C09107=1052.158,191.230,408.588,171.579,35.261,156.618
C09108=1052.153,190.981,408.612,171.577,35.259,156.618
C09109=1052.147,190.732,408.636,171.575,35.257,156.617
C09110=1052.140,190.448,408.663,171.573,35.253,156.616
C09111=1052.134,190.163,408.691,171.570,35.251,156.616
C09112=1052.127,189.880,408.719,171.567,35.248,156.615
C09113=1052.121,189.595,408.746,171.564,35.245,156.615
C09114=1052.114,189.346,408.770,171.562,35.242,156.614
C09115=1052.109,189.098,408.794,171.560,35.240,156.614
C09116=1052.102,188.849,408.818,171.558,35.237,156.613
C09117=1052.097,188.600,408.843,171.555,35.235,156.613
C09118=1052.091,188.352,408.866,171.553,35.232,156.612
C09119=1052.085,188.102,408.890,171.551,35.229,156.612
C09120=1052.079,187.854,408.914,171.549,35.227,156.611
C09121=1052.073,187.605,408.938,171.547,35.224,156.611
C09122=1052.067,187.356,408.962,171.543,35.222,156.611
C09123=1052.062,187.108,408.986,171.541,35.219,156.610
C09124=1052.055,186.859,409.010,171.539,35.217,156.610
C09125=1052.049,186.610,409.033,171.537,35.214,156.609
C09126=1052.044,186.361,409.058,171.535,35.212,156.609
C09127=1052.037,186.112,409.082,171.533,35.209,156.608
C09128=1052.032,185.864,409.106,171.530,35.206,156.608
C09129=1052.026,185.615,409.130,171.528,35.204,156.607
C09130=1052.021,185.365,409.153,171.526,35.201,156.607
C09131=1052.014,185.117,409.177,171.524,35.199,156.606
C09132=1052.009,184.869,409.201,171.522,35.196,156.606
C09133=1052.003,184.620,409.225,171.518,35.194,156.605
C09134=1051.997,184.371,409.248,171.516,35.191,156.605
C09135=1051.992,184.122,409.273,171.514,35.189,156.604
C09136=1051.985,183.873,409.297,171.512,35.187,156.604
C09137=1051.979,183.624,409.320,171.510,35.184,156.603
C09138=1051.973,183.375,409.344,171.508,35.182,156.603
C09139=1051.967,183.126,409.367,171.505,35.179,156.602
C09140=1051.961,182.878,409.390,171.503,35.177,156.602
C09141=1051.954,182.628,409.413,171.501,35.175,156.602
C09142=1051.948,182.380,409.437,171.499,35.172,156.601
C09143=1051.942,182.131,409.460,171.496,35.170,156.601
C09144=1051.935,181.883,409.484,171.494,35.167,156.600
C09145=1051.930,181.634,409.506,171.491,35.165,156.600
C09146=1051.923,181.385,409.530,171.489,35.163,156.599
C09147=1051.917,181.136,409.553,171.487,35.160,156.599
C09148=1051.911,180.888,409.577,171.485,35.158,156.599
C09149=1051.905,180.638,409.600,171.483,35.155,156.598
C09150=1051.899,180.390,409.624,171.481,35.154,156.598
C09151=1051.893,180.141,409.647,171.478,35.151,156.597
C09152=1051.886,179.892,409.671,171.476,35.149,156.597
C09153=1051.881,179.643,409.694,171.474,35.146,156.596
C09154=1051.875,179.395,409.718,171.472,35.144,156.596
C09155=1051.868,179.145,409.741,171.469,35.142,156.595
C09156=1051.862,178.896,409.763,171.467,35.139,156.595
C09157=1051.856,178.648,409.787,171.464,35.137,156.595
C09158=1051.849,178.399,409.810,171.462,35.134,156.594
C09159=1051.844,178.150,409.833,171.460,35.132,156.594
C09160=1051.838,177.901,409.857,171.458,35.130,156.593
C09161=1051.832,177.653,409.880,171.456,35.127,156.593
C09162=1051.825,177.404,409.904,171.454,35.125,156.592
C09163=1051.820,177.155,409.927,171.451,35.122,156.592
C09164=1051.814,176.906,409.950,171.449,35.120,156.592
C09165=1051.808,176.656,409.973,171.447,35.118,156.591
C09166=1051.801,176.408,409.996,171.445,35.115,156.591
C09167=1051.795,176.159,410.019,171.443,35.113,156.590
C09168=1051.789,175.910,410.042,171.441,35.111,156.590
C09169=1051.783,175.662,410.066,171.438,35.109,156.589
C09170=1051.777,175.413,410.089,171.436,35.106,156.589
C09171=1051.771,175.164,410.112,171.434,35.104,156.588
C09172=1051.765,174.915,410.135,171.432,35.102,156.588
C09173=1051.759,174.666,410.159,171.430,35.099,156.588
C09174=1051.752,174.381,410.185,171.427,35.096,156.587
C09175=1051.746,174.097,410.211,171.424,35.094,156.587
C09176=1051.739,173.813,410.237,171.422,35.091,156.586
C09177=1051.732,173.527,410.264,171.419,35.089,156.586
C09178=1051.725,173.279,410.286,171.417,35.086,156.585
C09179=1051.719,173.030,410.310,171.415,35.084,156.585
C09180=1051.714,172.781,410.333,171.413,35.081,156.584
C09181=1051.707,172.532,410.356,171.410,35.079,156.584
C09182=1051.702,172.283,410.379,171.408,35.077,156.583
C09183=1051.696,172.034,410.402,171.406,35.074,156.583
C09184=1051.689,171.786,410.424,171.404,35.072,156.583
C09185=1051.684,171.537,410.447,171.402,35.069,156.582
C09186=1051.678,171.288,410.470,171.400,35.067,156.582
C09187=1051.672,171.039,410.494,171.399,35.065,156.581
C09188=1051.666,170.791,410.517,171.396,35.062,156.581
C09189=1051.660,170.541,410.540,171.394,35.060,156.580
C09190=1051.653,170.292,410.563,171.392,35.058,156.580
C09191=1051.648,170.043,410.586,171.390,35.056,156.580
C09192=1051.642,169.795,410.608,171.388,35.053,156.579
C09193=1051.636,169.546,410.631,171.386,35.051,156.579
C09194=1051.630,169.297,410.654,171.383,35.049,156.578
C09195=1051.625,169.048,410.677,171.381,35.046,156.578
C09196=1051.618,168.799,410.700,171.379,35.044,156.577
C09197=1051.612,168.550,410.723,171.377,35.041,156.577
C09198=1051.607,168.302,410.746,171.375,35.039,156.577
C09199=1051.601,168.053,410.769,171.373,35.037,156.576
C09200=1051.595,167.804,410.791,171.370,35.034,156.576
C09201=1051.589,167.555,410.814,171.368,35.032,156.575
C09202=1051.583,167.306,410.837,171.366,35.030,156.575
C09203=1051.577,167.057,410.860,171.364,35.027,156.574
C09204=1051.572,166.808,410.883,171.362,35.025,156.574
C09205=1051.566,166.560,410.906,171.360,35.022,156.573
C09206=1051.559,166.311,410.928,171.358,35.020,156.573
C09207=1051.554,166.061,410.950,171.355,35.018,156.573
C09208=1051.548,165.813,410.973,171.353,35.015,156.572
C09209=1051.543,165.564,410.996,171.351,35.013,156.572
C09210=1051.537,165.315,411.019,171.350,35.011,156.571
C09211=1051.530,165.066,411.041,171.348,35.009,156.571
C09212=1051.525,164.817,411.064,171.346,35.006,156.570
C09213=1051.519,164.568,411.087,171.343,35.004,156.570
C09214=1051.513,164.319,411.109,171.341,35.002,156.570
C09215=1051.507,164.070,411.132,171.339,34.999,156.569
C09216=1051.501,163.821,411.155,171.337,34.997,156.569
C09217=1051.496,163.572,411.178,171.335,34.994,156.568
C09218=1051.490,163.324,411.201,171.333,34.992,156.568
C09219=1051.483,163.075,411.223,171.331,34.990,156.567
C09220=1051.478,162.825,411.245,171.328,34.987,156.567
C09221=1051.472,162.577,411.268,171.327,34.985,156.566
C09222=1051.466,162.328,411.291,171.325,34.983,156.566
C09223=1051.460,162.079,411.313,171.323,34.980,156.566
C09224=1051.455,161.830,411.336,171.321,34.978,156.565
C09225=1051.449,161.581,411.359,171.319,34.975,156.565
C09226=1051.444,161.332,411.381,171.317,34.974,156.564
C09227=1051.438,161.083,411.403,171.314,34.971,156.564
C09228=1051.432,160.834,411.426,171.312,34.969,156.564
C09229=1051.426,160.585,411.449,171.310,34.967,156.563
C09230=1051.420,160.336,411.470,171.308,34.964,156.563
C09231=1051.414,160.087,411.493,171.307,34.962,156.562
C09232=1051.408,159.839,411.516,171.305,34.960,156.562
C09233=1051.402,159.590,411.537,171.303,34.957,156.561
C09234=1051.396,159.341,411.560,171.300,34.955,156.561
C09235=1051.390,159.091,411.582,171.298,34.953,156.561
C09236=1051.384,158.843,411.605,171.296,34.951,156.560
C09237=1051.377,158.594,411.627,171.294,34.948,156.560
C09238=1051.371,158.309,411.652,171.292,34.946,156.559
C09239=1051.364,158.023,411.678,171.290,34.943,156.559
C09240=1051.357,157.739,411.703,171.288,34.941,156.558
C09241=1051.350,157.454,411.728,171.284,34.938,156.558
C09242=1051.344,157.205,411.751,171.283,34.937,156.558
C09243=1051.338,156.956,411.773,171.281,34.934,156.557
C09244=1051.332,156.707,411.795,171.279,34.932,156.557
C09245=1051.326,156.457,411.817,171.277,34.930,156.556
C09246=1051.320,156.209,411.840,171.275,34.927,156.556
C09247=1051.314,155.960,411.861,171.273,34.925,156.556
C09248=1051.308,155.711,411.884,171.270,34.923,156.555
C09249=1051.302,155.462,411.906,171.268,34.921,156.555
C09250=1051.296,155.213,411.927,171.266,34.918,156.554
C09251=1051.291,154.964,411.950,171.265,34.916,156.554
C09252=1051.284,154.715,411.972,171.263,34.914,156.554
C09253=1051.278,154.466,411.994,171.261,34.912,156.553
C09254=1051.273,154.217,412.016,171.259,34.909,156.553
C09255=1051.266,153.968,412.038,171.257,34.908,156.552
C09256=1051.260,153.719,412.060,171.254,34.905,156.552
C09257=1051.254,153.471,412.082,171.252,34.903,156.552
C09258=1051.248,153.221,412.103,171.251,34.901,156.551
C09259=1051.242,152.972,412.126,171.249,34.899,156.551
C09260=1051.236,152.723,412.148,171.247,34.896,156.550
C09261=1051.230,152.474,412.169,171.245,34.894,156.550
C09262=1051.224,152.225,412.192,171.243,34.892,156.550
C09263=1051.218,151.977,412.213,171.240,34.890,156.549
C09264=1051.213,151.727,412.235,171.238,34.887,156.549
C09265=1051.206,151.479,412.258,171.237,34.886,156.548
C09266=1051.200,151.230,412.279,171.235,34.883,156.548
C09267=1051.194,150.980,412.301,171.233,34.881,156.548
C09268=1051.188,150.731,412.323,171.231,34.879,156.547
C09269=1051.183,150.483,412.345,171.229,34.877,156.547
C09270=1051.176,150.234,412.367,171.227,34.874,156.546
C09271=1051.170,149.985,412.388,171.224,34.872,156.546
C09272=1051.164,149.735,412.410,171.223,34.870,156.546
C09273=1051.158,149.487,412.432,171.221,34.868,156.545
C09274=1051.152,149.238,412.454,171.219,34.866,156.545
C09275=1051.147,148.989,412.476,171.217,34.863,156.544
C09276=1051.140,148.740,412.498,171.215,34.862,156.544
C09277=1051.134,148.490,412.519,171.213,34.859,156.544
C09278=1051.129,148.242,412.540,171.212,34.857,156.543
C09279=1051.122,147.993,412.563,171.209,34.855,156.543
C09280=1051.116,147.744,412.584,171.207,34.853,156.542
C09281=1051.110,147.495,412.606,171.205,34.850,156.542
C09282=1051.104,147.246,412.627,171.203,34.848,156.542
C09283=1051.098,146.997,412.649,171.201,34.846,156.541
C09284=1051.092,146.748,412.671,171.200,34.844,156.541
C09285=1051.086,146.499,412.692,171.198,34.842,156.541
C09286=1051.080,146.250,412.714,171.196,34.840,156.540
C09287=1051.074,146.001,412.735,171.193,34.838,156.540
C09288=1051.068,145.752,412.757,171.191,34.836,156.539
C09289=1051.062,145.503,412.778,171.189,34.833,156.539
C09290=1051.056,145.253,412.800,171.188,34.831,156.539
C09291=1051.050,145.005,412.821,171.186,34.829,156.538
C09292=1051.044,144.756,412.843,171.184,34.827,156.538
C09293=1051.038,144.506,412.865,171.182,34.825,156.537
C09294=1051.032,144.258,412.886,171.180,34.823,156.537
C09295=1051.026,144.009,412.907,171.178,34.821,156.537
C09296=1051.020,143.760,412.929,171.176,34.819,156.536
C09297=1051.014,143.510,412.951,171.174,34.816,156.536
C09298=1051.007,143.262,412.971,171.172,34.814,156.536
C09299=1051.001,143.013,412.993,171.170,34.812,156.535
C09300=1050.995,142.764,413.015,171.169,34.810,156.535
C09301=1050.990,142.515,413.036,171.167,34.808,156.534
C09302=1050.982,142.229,413.061,171.165,34.805,156.534
C09303=1050.976,141.944,413.086,171.162,34.803,156.534
C09304=1050.969,141.659,413.110,171.160,34.800,156.533
C09305=1050.963,141.373,413.134,171.158,34.798,156.533
C09306=1050.956,141.124,413.156,171.156,34.796,156.532
C09307=1050.950,140.875,413.177,171.154,34.794,156.532
C09308=1050.945,140.626,413.199,171.152,34.791,156.531
C09309=1050.938,140.377,413.220,171.150,34.790,156.531
C09310=1050.932,140.129,413.241,171.149,34.787,156.531
C09311=1050.926,139.879,413.262,171.146,34.785,156.530
C09312=1050.920,139.630,413.284,171.144,34.783,156.530
C09313=1050.915,139.381,413.305,171.142,34.781,156.530
C09314=1050.908,139.132,413.326,171.140,34.779,156.529
C09315=1050.902,138.883,413.348,171.139,34.777,156.529
C09316=1050.896,138.634,413.368,171.137,34.774,156.528
C09317=1050.890,138.385,413.390,171.135,34.772,156.528
C09318=1050.884,138.136,413.411,171.133,34.771,156.528
C09319=1050.878,137.888,413.432,171.131,34.768,156.527
C09320=1050.872,137.638,413.453,171.129,34.766,156.527
C09321=1050.866,137.389,413.475,171.127,34.764,156.527
C09322=1050.860,137.140,413.496,171.125,34.762,156.526
C09323=1050.853,136.891,413.517,171.123,34.760,156.526
C09324=1050.848,136.642,413.537,171.122,34.758,156.525
C09325=1050.842,136.393,413.559,171.120,34.756,156.525
C09326=1050.835,136.144,413.580,171.118,34.753,156.525
C09327=1050.830,135.895,413.601,171.116,34.752,156.524
C09328=1050.823,135.646,413.622,171.114,34.750,156.524
C09329=1050.817,135.397,413.643,171.112,34.747,156.524
C09330=1050.811,135.148,413.664,171.110,34.745,156.523
C09331=1050.805,134.898,413.686,171.108,34.743,156.523
C09332=1050.799,134.650,413.705,171.107,34.741,156.522
C09333=1050.793,134.400,413.727,171.105,34.739,156.522
C09334=1050.787,134.152,413.748,171.103,34.737,156.522
C09335=1050.782,133.902,413.769,171.101,34.734,156.521
C09336=1050.775,133.654,413.790,171.100,34.733,156.521
C09337=1050.769,133.404,413.811,171.097,34.731,156.521
C09338=1050.763,133.156,413.832,171.095,34.729,156.520
C09339=1050.757,132.907,413.853,171.093,34.726,156.520
C09340=1050.751,132.657,413.874,171.092,34.724,156.519
C09341=1050.745,132.409,413.895,171.090,34.722,156.519
C09342=1050.739,132.159,413.916,171.088,34.720,156.519
C09343=1050.733,131.910,413.937,171.086,34.718,156.518
C09344=1050.727,131.661,413.957,171.085,34.716,156.518
C09345=1050.721,131.412,413.979,171.083,34.713,156.518
C09346=1050.715,131.163,413.999,171.080,34.712,156.517
C09347=1050.709,130.914,414.020,171.078,34.710,156.517
C09348=1050.702,130.665,414.041,171.077,34.708,156.517
C09349=1050.697,130.415,414.061,171.075,34.706,156.516
C09350=1050.690,130.167,414.082,171.073,34.704,156.516
C09351=1050.684,129.917,414.102,171.071,34.701,156.515
C09352=1050.678,129.669,414.124,171.069,34.699,156.515
C09353=1050.672,129.419,414.144,171.068,34.698,156.515
C09354=1050.665,129.171,414.165,171.066,34.696,156.514
C09355=1050.659,128.921,414.186,171.064,34.694,156.514
C09356=1050.653,128.672,414.206,171.061,34.691,156.514
C09357=1050.647,128.423,414.227,171.060,34.689,156.513
C09358=1050.641,128.174,414.248,171.058,34.687,156.513
C09359=1050.635,127.925,414.267,171.056,34.685,156.513
C09360=1050.628,127.676,414.289,171.054,34.684,156.512
C09361=1050.622,127.427,414.309,171.053,34.682,156.512
C09362=1050.616,127.177,414.329,171.051,34.679,156.512
C09363=1050.610,126.929,414.351,171.049,34.677,156.511
C09364=1050.604,126.679,414.371,171.048,34.675,156.511
C09365=1050.598,126.430,414.391,171.046,34.673,156.511
C09366=1050.591,126.145,414.415,171.043,34.671,156.510
C09367=1050.584,125.860,414.438,171.041,34.669,156.510
C09368=1050.577,125.574,414.462,171.039,34.666,156.509
C09369=1050.570,125.289,414.486,171.037,34.664,156.509
C09370=1050.564,125.039,414.507,171.035,34.662,156.508
C09371=1050.558,124.790,414.526,171.033,34.660,156.508
C09372=1050.551,124.541,414.547,171.032,34.658,156.508
C09373=1050.546,124.292,414.568,171.030,34.656,156.507
C09374=1050.539,124.043,414.588,171.028,34.654,156.507
C09375=1050.533,123.794,414.608,171.026,34.652,156.507
C09376=1050.528,123.545,414.629,171.024,34.650,156.506
C09377=1050.521,123.295,414.649,171.022,34.648,156.506
C09378=1050.515,123.047,414.670,171.020,34.645,156.506
C09379=1050.509,122.797,414.691,171.019,34.643,156.505
C09380=1050.503,122.548,414.711,171.017,34.642,156.505
C09381=1050.497,122.299,414.731,171.015,34.640,156.505
C09382=1050.491,122.050,414.752,171.014,34.638,156.504
C09383=1050.485,121.801,414.772,171.012,34.635,156.504
C09384=1050.478,121.552,414.793,171.009,34.633,156.503
C09385=1050.473,121.303,414.813,171.007,34.631,156.503
C09386=1050.467,121.054,414.833,171.006,34.629,156.503
C09387=1050.461,120.805,414.853,171.004,34.627,156.502
C09388=1050.455,120.556,414.873,171.002,34.625,156.502
C09389=1050.449,120.306,414.894,171.001,34.623,156.502
C09390=1050.443,120.057,414.914,170.999,34.621,156.501
C09391=1050.437,119.808,414.934,170.997,34.619,156.501
C09392=1050.431,119.559,414.955,170.996,34.617,156.501
C09393=1050.425,119.310,414.975,170.994,34.615,156.500
C09394=1050.419,119.061,414.995,170.991,34.613,156.500
C09395=1050.413,118.812,415.017,170.990,34.611,156.500
C09396=1050.407,118.563,415.037,170.988,34.608,156.499
C09397=1050.401,118.314,415.057,170.986,34.606,156.499
C09398=1050.394,118.065,415.077,170.985,34.605,156.498
C09399=1050.389,117.815,415.098,170.983,34.603,156.498
C09400=1050.383,117.567,415.118,170.981,34.600,156.498
C09401=1050.376,117.317,415.138,170.979,34.598,156.497
C09402=1050.371,117.068,415.158,170.978,34.596,156.497
C09403=1050.365,116.819,415.178,170.976,34.594,156.497
C09404=1050.359,116.570,415.198,170.973,34.592,156.496
C09405=1050.352,116.321,415.219,170.972,34.590,156.496
C09406=1050.347,116.072,415.239,170.970,34.588,156.495
C09407=1050.341,115.823,415.259,170.968,34.586,156.495
C09408=1050.335,115.573,415.279,170.967,34.584,156.495
C09409=1050.329,115.324,415.299,170.965,34.582,156.494
C09410=1050.324,115.075,415.319,170.963,34.580,156.494
C09411=1050.318,114.826,415.339,170.962,34.578,156.494
C09412=1050.311,114.577,415.360,170.960,34.575,156.493
C09413=1050.305,114.328,415.380,170.958,34.573,156.493
C09414=1050.300,114.079,415.400,170.957,34.571,156.493
C09415=1050.294,113.830,415.420,170.954,34.569,156.492
C09416=1050.287,113.580,415.440,170.952,34.567,156.492
C09417=1050.281,113.331,415.460,170.951,34.565,156.491
C09418=1050.276,113.082,415.480,170.949,34.563,156.491
C09419=1050.270,112.833,415.500,170.947,34.561,156.491
C09420=1050.263,112.584,415.520,170.946,34.559,156.490
C09421=1050.257,112.335,415.540,170.944,34.557,156.490
C09422=1050.251,112.086,415.560,170.942,34.555,156.490
C09423=1050.245,111.836,415.579,170.941,34.554,156.489
C09424=1050.239,111.587,415.599,170.939,34.551,156.489
C09425=1050.233,111.338,415.619,170.936,34.549,156.489
C09426=1050.227,111.089,415.639,170.935,34.547,156.488
C09427=1050.220,110.839,415.659,170.933,34.545,156.488
C09428=1050.214,110.591,415.679,170.931,34.543,156.488
C09429=1050.208,110.342,415.699,170.930,34.541,156.487
C09430=1050.201,110.056,415.721,170.928,34.539,156.487
C09431=1050.194,109.770,415.744,170.926,34.537,156.487
C09432=1050.187,109.484,415.766,170.924,34.534,156.486
C09433=1050.180,109.198,415.789,170.922,34.532,156.486
C09434=1050.173,108.950,415.809,170.920,34.530,156.485
C09435=1050.167,108.701,415.829,170.919,34.529,156.485
C09436=1050.162,108.452,415.848,170.916,34.526,156.485
C09437=1050.155,108.202,415.868,170.914,34.524,156.484
C09438=1050.149,107.953,415.888,170.913,34.522,156.484
C09439=1050.143,107.704,415.907,170.911,34.520,156.484
C09440=1050.137,107.455,415.927,170.909,34.518,156.483
C09441=1050.131,107.206,415.947,170.908,34.516,156.483
C09442=1050.124,106.956,415.966,170.906,34.514,156.483
C09443=1050.118,106.708,415.986,170.904,34.513,156.482
C09444=1050.113,106.458,416.006,170.903,34.511,156.482
C09445=1050.107,106.209,416.026,170.901,34.509,156.482
C09446=1050.101,105.960,416.045,170.899,34.506,156.481
C09447=1050.094,105.711,416.064,170.897,34.504,156.481
C09448=1050.088,105.462,416.084,170.895,34.502,156.481
C09449=1050.082,105.212,416.104,170.893,34.500,156.480
C09450=1050.076,104.964,416.124,170.892,34.498,156.480
C09451=1050.070,104.714,416.143,170.890,34.497,156.480
C09452=1050.064,104.465,416.163,170.888,34.495,156.479
C09453=1050.057,104.216,416.182,170.887,34.493,156.479
C09454=1050.051,103.967,416.202,170.885,34.491,156.479
C09455=1050.046,103.717,416.221,170.884,34.488,156.478
C09456=1050.040,103.468,416.241,170.882,34.486,156.478
C09457=1050.034,103.219,416.260,170.880,34.484,156.477
C09458=1050.028,102.970,416.280,170.878,34.482,156.477
C09459=1050.022,102.721,416.299,170.876,34.481,156.477
C09460=1050.016,102.472,416.319,170.874,34.479,156.476
C09461=1050.009,102.222,416.338,170.873,34.477,156.476
C09462=1050.003,101.973,416.358,170.871,34.475,156.476
C09463=1049.998,101.724,416.378,170.869,34.472,156.475
C09464=1049.991,101.475,416.397,170.868,34.470,156.475
C09465=1049.985,101.226,416.416,170.866,34.468,156.475
C09466=1049.979,100.977,416.436,170.864,34.466,156.474
C09467=1049.973,100.728,416.455,170.863,34.464,156.474
C09468=1049.967,100.479,416.474,170.861,34.463,156.474
C09469=1049.961,100.230,416.494,170.860,34.461,156.473
C09470=1049.955,99.980,416.514,170.857,34.459,156.473
C09471=1049.948,99.731,416.532,170.855,34.457,156.473
C09472=1049.942,99.482,416.552,170.854,34.455,156.472
C09473=1049.936,99.233,416.571,170.852,34.453,156.472
C09474=1049.930,98.983,416.590,170.850,34.451,156.472
C09475=1049.923,98.735,416.610,170.849,34.449,156.471
C09476=1049.918,98.485,416.629,170.847,34.447,156.471
C09477=1049.911,98.236,416.647,170.845,34.445,156.471
C09478=1049.905,97.986,416.667,170.844,34.443,156.470
C09479=1049.899,97.737,416.687,170.842,34.441,156.470
C09480=1049.893,97.488,416.706,170.840,34.439,156.470
C09481=1049.887,97.239,416.725,170.839,34.437,156.469
C09482=1049.881,96.989,416.744,170.836,34.436,156.469
C09483=1049.875,96.741,416.764,170.834,34.434,156.469
C09484=1049.868,96.492,416.782,170.833,34.432,156.468
C09485=1049.862,96.242,416.801,170.831,34.429,156.468
C09486=1049.856,95.993,416.820,170.830,34.427,156.468
C09487=1049.850,95.744,416.840,170.828,34.425,156.467
C09488=1049.844,95.495,416.859,170.826,34.423,156.467
C09489=1049.838,95.246,416.878,170.825,34.421,156.467
C09490=1049.832,94.996,416.897,170.823,34.419,156.466
C09491=1049.826,94.747,416.916,170.821,34.418,156.466
C09492=1049.820,94.498,416.936,170.820,34.416,156.466
C09493=1049.813,94.249,416.954,170.818,34.414,156.465
C09494=1049.808,94.014,416.972,170.817,34.412,156.465
C09495=1049.802,93.780,416.990,170.814,34.410,156.465
C09496=1049.797,93.545,417.008,170.813,34.408,156.464
C09497=1049.790,93.311,417.026,170.811,34.407,156.464
C09498=1049.784,93.076,417.044,170.809,34.405,156.464
C09499=1049.779,92.842,417.063,170.808,34.403,156.463
C09500=1049.773,92.608,417.080,170.806,34.401,156.463
C09501=1049.768,92.374,417.098,170.805,34.399,156.463
C09502=1049.761,92.124,417.117,170.803,34.397,156.462
C09503=1049.756,91.875,417.136,170.802,34.395,156.462
C09504=1049.749,91.626,417.155,170.800,34.393,156.462
C09505=1049.744,91.376,417.174,170.798,34.391,156.461
C09506=1049.737,91.127,417.193,170.797,34.389,156.461
C09507=1049.731,90.878,417.212,170.795,34.387,156.461
C09508=1049.725,90.629,417.231,170.793,34.385,156.460
C09509=1049.719,90.379,417.250,170.791,34.383,156.460
C09510=1049.711,90.064,417.274,170.789,34.381,156.460
C09511=1049.703,89.749,417.298,170.787,34.378,156.459
C09512=1049.695,89.433,417.321,170.785,34.376,156.459
C09513=1049.687,89.119,417.345,170.783,34.374,156.458
C09514=1049.681,88.870,417.364,170.781,34.372,156.458
C09515=1049.675,88.620,417.383,170.779,34.370,156.458
C09516=1049.669,88.371,417.401,170.778,34.368,156.457
C09517=1049.663,88.122,417.420,170.776,34.366,156.457
C09518=1049.656,87.873,417.439,170.774,34.364,156.457
C09519=1049.650,87.624,417.458,170.773,34.362,156.456
C09520=1049.644,87.374,417.476,170.770,34.360,156.456
C09521=1049.638,87.125,417.495,170.769,34.358,156.456
C09522=1049.631,86.876,417.513,170.767,34.356,156.456
C09523=1049.626,86.626,417.532,170.765,34.354,156.455
C09524=1049.619,86.377,417.551,170.764,34.352,156.455
C09525=1049.613,86.128,417.570,170.762,34.350,156.455
C09526=1049.606,85.879,417.588,170.760,34.349,156.454
C09527=1049.601,85.629,417.608,170.759,34.347,156.454
C09528=1049.594,85.380,417.626,170.757,34.345,156.454
C09529=1049.588,85.131,417.644,170.756,34.343,156.453
C09530=1049.582,84.881,417.663,170.754,34.341,156.453
C09531=1049.577,84.633,417.682,170.752,34.339,156.453
C09532=1049.570,84.384,417.700,170.751,34.337,156.452
C09533=1049.564,84.134,417.719,170.749,34.335,156.452
C09534=1049.557,83.885,417.738,170.746,34.333,156.452
C09535=1049.551,83.636,417.756,170.745,34.331,156.451
C09536=1049.546,83.386,417.775,170.743,34.329,156.451
C09537=1049.539,83.137,417.793,170.742,34.327,156.451
C09538=1049.533,82.888,417.812,170.740,34.325,156.450
C09539=1049.527,82.638,417.830,170.738,34.323,156.450
C09540=1049.521,82.390,417.848,170.737,34.321,156.450
C09541=1049.515,82.140,417.868,170.735,34.319,156.449
C09542=1049.509,81.891,417.886,170.733,34.318,156.449
C09543=1049.502,81.642,417.905,170.732,34.316,156.449
C09544=1049.496,81.392,417.923,170.730,34.314,156.448
C09545=1049.490,81.143,417.941,170.729,34.312,156.448
C09546=1049.484,80.894,417.961,170.727,34.310,156.448
C09547=1049.479,80.645,417.978,170.724,34.308,156.447
C09548=1049.472,80.396,417.997,170.723,34.306,156.447
C09549=1049.466,80.146,418.016,170.721,34.304,156.447
C09550=1049.459,79.897,418.034,170.720,34.302,156.446
C09551=1049.454,79.647,418.053,170.718,34.300,156.446
C09552=1049.448,79.399,418.071,170.716,34.298,156.446
C09553=1049.442,79.150,418.090,170.715,34.296,156.445
C09554=1049.436,78.900,418.108,170.713,34.294,156.445
C09555=1049.429,78.651,418.126,170.712,34.292,156.445
C09556=1049.423,78.401,418.144,170.710,34.290,156.444
C09557=1049.417,78.152,418.163,170.708,34.288,156.444
C09558=1049.410,77.866,418.184,170.706,34.286,156.444
C09559=1049.403,77.581,418.205,170.705,34.285,156.443
C09560=1049.396,77.296,418.226,170.703,34.282,156.443
C09561=1049.388,77.009,418.247,170.700,34.280,156.443
C09562=1049.382,76.760,418.265,170.698,34.278,156.442
C09563=1049.376,76.511,418.283,170.697,34.276,156.442
C09564=1049.370,76.262,418.301,170.695,34.274,156.442
C09565=1049.364,76.012,418.320,170.693,34.272,156.441
C09566=1049.358,75.763,418.338,170.692,34.270,156.441
C09567=1049.351,75.514,418.356,170.690,34.268,156.441
C09568=1049.346,75.265,418.374,170.688,34.267,156.440
C09569=1049.339,75.015,418.393,170.687,34.265,156.440
C09570=1049.333,74.766,418.411,170.685,34.263,156.440
C09571=1049.327,74.517,418.429,170.684,34.261,156.439
C09572=1049.321,74.267,418.447,170.682,34.259,156.439
C09573=1049.315,74.018,418.465,170.680,34.257,156.439
C09574=1049.309,73.769,418.483,170.679,34.255,156.438
C09575=1049.302,73.520,418.502,170.677,34.253,156.438
C09576=1049.295,73.270,418.519,170.675,34.251,156.438
C09577=1049.290,73.022,418.538,170.673,34.250,156.437
C09578=1049.284,72.772,418.556,170.671,34.248,156.437
C09579=1049.277,72.523,418.574,170.670,34.246,156.437
C09580=1049.271,72.273,418.592,170.668,34.244,156.436
C09581=1049.265,72.024,418.610,170.666,34.242,156.436
C09582=1049.259,71.775,418.628,170.665,34.240,156.436
C09583=1049.253,71.525,418.646,170.663,34.238,156.436
C09584=1049.247,71.277,418.665,170.662,34.237,156.435
C09585=1049.241,71.027,418.683,170.660,34.235,156.435
C09586=1049.234,70.778,418.700,170.658,34.233,156.435
C09587=1049.228,70.528,418.719,170.657,34.231,156.434
C09588=1049.222,70.279,418.736,170.655,34.229,156.434
C09589=1049.216,70.030,418.754,170.653,34.227,156.434
C09590=1049.210,69.781,418.773,170.652,34.225,156.433
C09591=1049.204,69.532,418.790,170.650,34.223,156.433
C09592=1049.198,69.282,418.808,170.648,34.221,156.433
C09593=1049.191,69.033,418.826,170.646,34.220,156.432
C09594=1049.185,68.783,418.844,170.644,34.218,156.432
C09595=1049.179,68.534,418.862,170.643,34.216,156.432
C09596=1049.173,68.285,418.880,170.641,34.214,156.431
C09597=1049.166,68.036,418.898,170.640,34.212,156.431
C09598=1049.160,67.787,418.915,170.638,34.210,156.431
C09599=1049.154,67.537,418.933,170.636,34.208,156.431
C09600=1049.148,67.288,418.952,170.635,34.206,156.430
C09601=1049.142,67.039,418.969,170.633,34.204,156.430
C09602=1049.135,66.789,418.987,170.631,34.203,156.430
C09603=1049.129,66.540,419.005,170.630,34.201,156.429
C09604=1049.123,66.291,419.022,170.628,34.199,156.429
C09605=1049.117,66.042,419.040,170.627,34.197,156.429
C09606=1049.111,65.792,419.058,170.625,34.195,156.428
C09607=1049.105,65.543,419.076,170.623,34.193,156.428
C09608=1049.098,65.293,419.093,170.621,34.191,156.428
C09609=1049.092,65.044,419.112,170.619,34.190,156.427
C09610=1049.086,64.795,419.129,170.617,34.188,156.427
C09611=1049.079,64.546,419.147,170.616,34.186,156.427
C09612=1049.073,64.296,419.165,170.614,34.184,156.427
C09613=1049.068,64.047,419.182,170.613,34.182,156.426
C09614=1049.061,63.798,419.200,170.611,34.180,156.426
C09615=1049.055,63.548,419.217,170.609,34.179,156.426
C09616=1049.048,63.298,419.235,170.608,34.177,156.425
C09617=1049.042,63.049,419.252,170.606,34.175,156.425
C09618=1049.035,62.800,419.270,170.604,34.173,156.425
C09619=1049.028,62.551,419.288,170.603,34.171,156.424
C09620=1049.023,62.302,419.305,170.601,34.169,156.424
C09621=1049.016,62.053,419.323,170.599,34.167,156.424
C09622=1049.009,61.767,419.343,170.597,34.165,156.424
C09623=1049.002,61.481,419.363,170.596,34.164,156.423
C09624=1048.994,61.194,419.383,170.594,34.162,156.423
C09625=1048.987,60.908,419.403,170.592,34.160,156.423
C09626=1048.981,60.660,419.420,170.589,34.158,156.422
C09627=1048.975,60.410,419.438,170.588,34.156,156.422
C09628=1048.968,60.160,419.455,170.586,34.154,156.422
C09629=1048.962,59.912,419.472,170.584,34.152,156.421
C09630=1048.956,59.662,419.490,170.583,34.150,156.421
C09631=1048.949,59.413,419.507,170.581,34.148,156.421
C09632=1048.943,59.163,419.525,170.579,34.146,156.420
C09633=1048.937,58.914,419.542,170.578,34.145,156.420
C09634=1048.930,58.665,419.559,170.576,34.143,156.420
C09635=1048.924,58.416,419.577,170.574,34.141,156.420
C09636=1048.917,58.166,419.595,170.573,34.139,156.419
C09637=1048.912,57.917,419.612,170.571,34.137,156.419
C09638=1048.905,57.668,419.629,170.569,34.136,156.419
C09639=1048.899,57.419,419.647,170.568,34.134,156.418
C09640=1048.893,57.169,419.664,170.566,34.132,156.418
C09641=1048.886,56.920,419.681,170.565,34.130,156.418
C09642=1048.881,56.670,419.699,170.563,34.128,156.417
C09643=1048.874,56.421,419.716,170.561,34.127,156.417
C09644=1048.868,56.172,419.733,170.560,34.125,156.417
C09645=1048.861,55.922,419.751,170.557,34.123,156.417
C09646=1048.855,55.673,419.768,170.555,34.121,156.416
C09647=1048.849,55.424,419.786,170.554,34.120,156.416
C09648=1048.843,55.175,419.803,170.552,34.118,156.416
C09649=1048.836,54.925,419.819,170.550,34.116,156.415
C09650=1048.831,54.676,419.837,170.549,34.114,156.415
C09651=1048.824,54.426,419.854,170.547,34.112,156.415
C09652=1048.818,54.177,419.872,170.546,34.110,156.414
C09653=1048.811,53.928,419.889,170.544,34.109,156.414
C09654=1048.805,53.679,419.905,170.542,34.107,156.414
C09655=1048.799,53.429,419.923,170.541,34.105,156.414
C09656=1048.793,53.180,419.940,170.539,34.103,156.413
C09657=1048.786,52.931,419.958,170.537,34.101,156.413
C09658=1048.781,52.682,419.975,170.536,34.099,156.413
C09659=1048.774,52.432,419.992,170.534,34.097,156.412
C09660=1048.769,52.183,420.009,170.532,34.095,156.412
C09661=1048.762,51.933,420.027,170.531,34.093,156.412
C09662=1048.755,51.684,420.044,170.529,34.092,156.411
C09663=1048.750,51.434,420.061,170.528,34.090,156.411
C09664=1048.743,51.185,420.078,170.525,34.088,156.411
C09665=1048.737,50.936,420.095,170.523,34.086,156.411
C09666=1048.731,50.686,420.112,170.522,34.084,156.410
C09667=1048.725,50.438,420.129,170.520,34.083,156.410
C09668=1048.718,50.188,420.146,170.518,34.081,156.410
C09669=1048.713,49.938,420.163,170.517,34.079,156.409
C09670=1048.706,49.689,420.181,170.515,34.077,156.409
C09671=1048.700,49.440,420.197,170.513,34.075,156.409
C09672=1048.694,49.190,420.215,170.512,34.073,156.408
C09673=1048.688,48.941,420.232,170.510,34.072,156.408
C09674=1048.682,48.692,420.249,170.509,34.070,156.408
C09675=1048.676,48.442,420.266,170.507,34.068,156.408
C09676=1048.670,48.193,420.283,170.505,34.066,156.407
C09677=1048.663,47.944,420.301,170.504,34.064,156.407
C09678=1048.657,47.694,420.317,170.502,34.063,156.407
C09679=1048.651,47.446,420.334,170.500,34.061,156.406
C09680=1048.645,47.196,420.351,170.499,34.059,156.406
C09681=1048.639,46.947,420.368,170.497,34.057,156.406
C09682=1048.633,46.698,420.385,170.495,34.055,156.405
C09683=1048.626,46.448,420.402,170.494,34.053,156.405
C09684=1048.621,46.199,420.419,170.491,34.051,156.405
C09685=1048.614,45.949,420.436,170.490,34.049,156.405
C09686=1048.607,45.663,420.456,170.488,34.047,156.404
C09687=1048.601,45.376,420.475,170.486,34.045,156.404
C09688=1048.593,45.091,420.495,170.484,34.043,156.403
C09689=1048.586,44.804,420.514,170.482,34.041,156.403
C09690=1048.581,44.555,420.531,170.480,34.039,156.403
C09691=1048.575,44.306,420.548,170.479,34.037,156.402
C09692=1048.568,44.056,420.565,170.477,34.035,156.402
C09693=1048.562,43.807,420.581,170.476,34.033,156.402
C09694=1048.556,43.558,420.599,170.474,34.031,156.402
C09695=1048.550,43.308,420.615,170.472,34.030,156.401
C09696=1048.544,43.059,420.632,170.471,34.028,156.401
C09697=1048.537,42.809,420.649,170.469,34.026,156.401
C09698=1048.531,42.560,420.666,170.467,34.024,156.400
C09699=1048.525,42.311,420.682,170.466,34.023,156.400
C09700=1048.518,42.061,420.699,170.464,34.021,156.400
C09701=1048.512,41.812,420.716,170.462,34.019,156.400
C09702=1048.506,41.563,420.732,170.461,34.017,156.399
C09703=1048.499,41.313,420.749,170.459,34.015,156.399
C09704=1048.494,41.064,420.766,170.457,34.013,156.399
C09705=1048.488,40.814,420.782,170.455,34.012,156.398
C09706=1048.481,40.565,420.800,170.453,34.010,156.398
C09707=1048.475,40.316,420.816,170.451,34.008,156.398
C09708=1048.469,40.066,420.832,170.450,34.006,156.397
C09709=1048.462,39.817,420.850,170.448,34.005,156.397
C09710=1048.457,39.567,420.866,170.446,34.003,156.397
C09711=1048.451,39.318,420.882,170.445,34.001,156.397
C09712=1048.444,39.069,420.899,170.443,33.999,156.396
C09713=1048.438,38.819,420.916,170.441,33.997,156.396
C09714=1048.432,38.570,420.932,170.440,33.995,156.396
C09715=1048.426,38.321,420.949,170.438,33.993,156.395
C09716=1048.420,38.072,420.965,170.436,33.992,156.395
C09717=1048.413,37.822,420.982,170.435,33.990,156.395
C09718=1048.407,37.572,420.998,170.433,33.988,156.395
C09719=1048.401,37.324,421.015,170.431,33.986,156.394
C09720=1048.394,37.074,421.032,170.430,33.985,156.394
C09721=1048.388,36.824,421.048,170.428,33.983,156.394
C09722=1048.382,36.575,421.064,170.426,33.982,156.394
C09723=1048.375,36.326,421.081,170.425,33.980,156.393
C09724=1048.369,36.076,421.097,170.423,33.978,156.393
C09725=1048.363,35.827,421.114,170.421,33.976,156.393
C09726=1048.357,35.578,421.130,170.420,33.974,156.392
C09727=1048.350,35.328,421.146,170.418,33.972,156.392
C09728=1048.344,35.078,421.163,170.416,33.971,156.392
C09729=1048.338,34.830,421.180,170.414,33.969,156.392
C09730=1048.332,34.581,421.195,170.412,33.968,156.391
C09731=1048.325,34.331,421.212,170.410,33.966,156.391
C09732=1048.319,34.081,421.228,170.408,33.964,156.391
C09733=1048.313,33.832,421.244,170.407,33.962,156.391
C09734=1048.307,33.583,421.261,170.405,33.960,156.390
C09735=1048.300,33.333,421.277,170.403,33.958,156.390
C09736=1048.294,33.083,421.293,170.402,33.957,156.390
C09737=1048.288,32.835,421.310,170.400,33.955,156.389
C09738=1048.282,32.585,421.326,170.398,33.954,156.389
C09739=1048.275,32.335,421.343,170.397,33.952,156.389
C09740=1048.269,32.086,421.359,170.395,33.950,156.389
C09741=1048.262,31.837,421.375,170.393,33.948,156.388
C09742=1048.257,31.588,421.391,170.392,33.946,156.388
C09743=1048.251,31.338,421.407,170.390,33.944,156.388
C09744=1048.244,31.088,421.424,170.388,33.943,156.387
C09745=1048.238,30.839,421.440,170.387,33.941,156.387
C09746=1048.231,30.590,421.456,170.385,33.939,156.387
C09747=1048.225,30.340,421.472,170.383,33.938,156.387
C09748=1048.219,30.091,421.488,170.382,33.936,156.386
C09749=1048.214,29.842,421.505,170.380,33.934,156.386
C09750=1048.206,29.556,421.523,170.378,33.932,156.386
C09751=1048.199,29.269,421.542,170.376,33.930,156.385
C09752=1048.191,28.983,421.560,170.374,33.928,156.385
C09753=1048.185,28.696,421.580,170.372,33.926,156.385
C09754=1048.178,28.447,421.595,170.370,33.924,156.385
C09755=1048.172,28.197,421.611,170.368,33.922,156.384
C09756=1048.166,27.948,421.627,170.366,33.921,156.384
C09757=1048.159,27.698,421.643,170.364,33.919,156.384
C09758=1048.153,27.449,421.659,170.363,33.917,156.383
C09759=1048.146,27.200,421.675,170.361,33.916,156.383
C09760=1048.140,26.951,421.691,170.359,33.914,156.383
C09761=1048.135,26.701,421.708,170.357,33.912,156.383
C09762=1048.128,26.452,421.723,170.356,33.910,156.382
C09763=1048.122,26.203,421.740,170.354,33.909,156.382
C09764=1048.115,25.953,421.756,170.352,33.907,156.382
C09765=1048.109,25.703,421.771,170.351,33.906,156.382
C09766=1048.103,25.454,421.787,170.349,33.904,156.381
C09767=1048.096,25.205,421.803,170.347,33.902,156.381
C09768=1048.090,24.955,421.819,170.345,33.900,156.381
C09769=1048.084,24.706,421.835,170.344,33.898,156.380
C09770=1048.078,24.457,421.851,170.342,33.897,156.380
C09771=1048.072,24.207,421.867,170.340,33.895,156.380
C09772=1048.065,23.957,421.883,170.339,33.894,156.380
C09773=1048.059,23.708,421.899,170.337,33.892,156.379
C09774=1048.052,23.459,421.915,170.335,33.890,156.379
C09775=1048.047,23.209,421.930,170.333,33.888,156.379
C09776=1048.040,22.960,421.946,170.332,33.887,156.379
C09777=1048.034,22.711,421.962,170.330,33.885,156.378
C09778=1048.028,22.461,421.978,170.328,33.884,156.378
C09779=1048.021,22.212,421.994,170.327,33.882,156.378
C09780=1048.016,21.962,422.010,170.325,33.880,156.378
C09781=1048.009,21.713,422.025,170.323,33.878,156.377
C09782=1048.003,21.464,422.042,170.321,33.876,156.377
C09783=1047.997,21.214,422.056,170.320,33.875,156.377
C09784=1047.990,20.964,422.073,170.318,33.873,156.377
C09785=1047.983,20.715,422.089,170.316,33.872,156.376
C09786=1047.977,20.466,422.105,170.315,33.870,156.376
C09787=1047.971,20.216,422.120,170.312,33.868,156.376
C09788=1047.965,19.967,422.136,170.310,33.866,156.375
C09789=1047.958,19.718,422.152,170.308,33.865,156.375
C09790=1047.953,19.468,422.167,170.307,33.863,156.375
C09791=1047.946,19.219,422.183,170.305,33.862,156.375
C09792=1047.940,18.969,422.199,170.303,33.860,156.374
C09793=1047.934,18.720,422.214,170.301,33.858,156.374
C09794=1047.928,18.470,422.231,170.300,33.856,156.374
C09795=1047.921,18.221,422.245,170.298,33.855,156.374
C09796=1047.915,17.972,422.261,170.296,33.853,156.373
C09797=1047.909,17.722,422.277,170.294,33.852,156.373
C09798=1047.902,17.473,422.292,170.293,33.850,156.373
C09799=1047.896,17.223,422.309,170.291,33.848,156.373
C09800=1047.890,16.974,422.324,170.289,33.846,156.372
C09801=1047.883,16.725,422.339,170.288,33.845,156.372
C09802=1047.878,16.475,422.355,170.286,33.843,156.372
C09803=1047.871,16.226,422.370,170.284,33.841,156.372
C09804=1047.865,15.976,422.386,170.282,33.839,156.371
C09805=1047.859,15.727,422.402,170.281,33.838,156.371
C09806=1047.852,15.477,422.417,170.279,33.836,156.371
C09807=1047.846,15.228,422.433,170.277,33.835,156.371
C09808=1047.840,14.978,422.448,170.275,33.833,156.370
C09809=1047.833,14.729,422.463,170.274,33.831,156.370
C09810=1047.828,14.479,422.479,170.272,33.830,156.370
C09811=1047.821,14.230,422.495,170.270,33.828,156.370
C09812=1047.815,13.980,422.510,170.268,33.827,156.369
C09813=1047.809,13.731,422.526,170.267,33.825,156.369
C09814=1047.801,13.446,422.544,170.265,33.823,156.369
C09815=1047.794,13.161,422.561,170.262,33.821,156.369
C09816=1047.787,12.876,422.579,170.260,33.819,156.368
C09817=1047.779,12.591,422.596,170.258,33.818,156.368
C09818=1047.773,12.341,422.611,170.257,33.816,156.368
C09819=1047.766,12.091,422.626,170.255,33.815,156.368
C09820=1047.760,11.843,422.641,170.253,33.813,156.367
C09821=1047.754,11.593,422.656,170.251,33.811,156.367
C09822=1047.747,11.344,422.671,170.250,33.810,156.367
C09823=1047.741,11.094,422.688,170.248,33.808,156.367
C09824=1047.735,10.845,422.702,170.246,33.806,156.366
C09825=1047.728,10.596,422.718,170.244,33.805,156.366
C09826=1047.722,10.346,422.733,170.241,33.803,156.366
C09827=1047.716,10.096,422.748,170.240,33.802,156.366
C09828=1047.709,9.847,422.763,170.238,33.800,156.365
C09829=1047.703,9.598,422.779,170.236,33.798,156.365
C09830=1047.697,9.348,422.794,170.234,33.797,156.365
C09831=1047.691,9.098,422.809,170.233,33.796,156.365
C09832=1047.684,8.849,422.825,170.231,33.794,156.364
C09833=1047.677,8.599,422.840,170.229,33.792,156.364
C09834=1047.671,8.350,422.855,170.227,33.791,156.364
C09835=1047.665,8.101,422.869,170.225,33.789,156.364
C09836=1047.659,7.852,422.885,170.224,33.787,156.363
C09837=1047.652,7.602,422.900,170.222,33.786,156.363
C09838=1047.647,7.352,422.915,170.220,33.784,156.363
C09839=1047.640,7.103,422.930,170.218,33.783,156.363
C09840=1047.633,6.853,422.946,170.217,33.781,156.363
C09841=1047.627,6.604,422.961,170.215,33.779,156.362
C09842=1047.621,6.354,422.976,170.213,33.778,156.362
C09843=1047.614,6.105,422.991,170.211,33.777,156.362
C09844=1047.609,5.856,423.005,170.209,33.774,156.362
C09845=1047.602,5.607,423.021,170.208,33.773,156.361
C09846=1047.595,5.357,423.036,170.206,33.771,156.361
C09847=1047.589,5.107,423.051,170.204,33.770,156.361
C09848=1047.583,4.857,423.067,170.202,33.768,156.361
C09849=1047.577,4.608,423.081,170.200,33.766,156.360
C09850=1047.571,4.359,423.096,170.199,33.765,156.360
C09851=1047.565,4.110,423.112,170.197,33.764,156.360
C09852=1047.558,3.860,423.127,170.195,33.762,156.360
C09853=1047.552,3.610,423.142,170.193,33.760,156.359
C09854=1047.545,3.361,423.157,170.191,33.759,156.359
C09855=1047.540,3.112,423.171,170.190,33.757,156.359
C09856=1047.533,2.862,423.186,170.188,33.756,156.359
C09857=1047.527,2.612,423.201,170.186,33.754,156.359
C09858=1047.521,2.363,423.216,170.184,33.752,156.358
C09859=1047.514,2.113,423.231,170.182,33.751,156.358
C09860=1047.509,1.864,423.247,170.181,33.749,156.358
C09861=1047.502,1.615,423.262,170.179,33.747,156.358
C09862=1047.496,1.365,423.277,170.177,33.746,156.357
C09863=1047.490,1.115,423.292,170.175,33.745,156.357
C09864=1047.484,0.866,423.306,170.173,33.743,156.357
C09865=1047.477,0.617,423.321,170.172,33.741,156.357
C09866=1047.471,0.367,423.336,170.170,33.740,156.356
C09867=1047.465,0.117,423.351,170.168,33.738,156.356
C09868=1047.459,-0.131,423.366,170.166,33.736,156.356
C09869=1047.453,-0.381,423.381,170.164,33.735,156.356
C09870=1047.446,-0.631,423.396,170.163,33.733,156.355
C09871=1047.440,-0.880,423.410,170.161,33.732,156.355
C09872=1047.434,-1.129,423.425,170.159,33.730,156.355
C09873=1047.428,-1.379,423.440,170.157,33.728,156.355
C09874=1047.421,-1.629,423.455,170.155,33.727,156.354
C09875=1047.415,-1.878,423.470,170.154,33.725,156.354
C09876=1047.409,-2.127,423.484,170.152,33.724,156.354
C09877=1047.403,-2.377,423.499,170.150,33.722,156.354
C09878=1047.396,-2.661,423.516,170.147,33.720,156.353
C09879=1047.390,-2.943,423.533,170.145,33.718,156.353
C09880=1047.382,-3.226,423.549,170.143,33.717,156.353
C09881=1047.375,-3.509,423.566,170.141,33.715,156.353
C09882=1047.369,-3.760,423.581,170.139,33.713,156.352
C09883=1047.363,-4.008,423.595,170.137,33.712,156.352
C09884=1047.356,-4.258,423.610,170.135,33.710,156.352
C09885=1047.350,-4.507,423.625,170.133,33.709,156.352
C09886=1047.343,-4.757,423.640,170.131,33.707,156.352
C09887=1047.338,-5.006,423.654,170.130,33.706,156.351
C09888=1047.331,-5.256,423.668,170.128,33.704,156.351
C09889=1047.324,-5.506,423.683,170.126,33.703,156.351
C09890=1047.318,-5.755,423.698,170.124,33.702,156.351
C09891=1047.312,-6.004,423.712,170.122,33.700,156.351
C09892=1047.305,-6.254,423.727,170.120,33.699,156.350
C09893=1047.299,-6.504,423.741,170.118,33.697,156.350
C09894=1047.293,-6.753,423.755,170.117,33.695,156.350
C09895=1047.286,-7.002,423.770,170.115,33.694,156.350
C09896=1047.280,-7.252,423.785,170.113,33.693,156.349
C09897=1047.274,-7.501,423.799,170.111,33.691,156.349
C09898=1047.268,-7.751,423.813,170.109,33.690,156.349
C09899=1047.261,-8.000,423.828,170.107,33.688,156.349
C09900=1047.255,-8.250,423.842,170.105,33.686,156.349
C09901=1047.249,-8.500,423.857,170.104,33.685,156.348
C09902=1047.242,-8.749,423.871,170.102,33.684,156.348
C09903=1047.236,-8.999,423.885,170.100,33.682,156.348
C09904=1047.230,-9.248,423.900,170.098,33.681,156.348
C09905=1047.223,-9.498,423.915,170.096,33.679,156.348
C09906=1047.217,-9.747,423.928,170.094,33.677,156.347
C09907=1047.211,-9.997,423.943,170.092,33.676,156.347
C09908=1047.205,-10.246,423.958,170.091,33.675,156.347
C09909=1047.198,-10.496,423.971,170.089,33.673,156.347
C09910=1047.192,-10.745,423.986,170.087,33.672,156.347
C09911=1047.186,-10.994,424.001,170.085,33.670,156.346
C09912=1047.179,-11.244,424.014,170.083,33.669,156.346
C09913=1047.174,-11.493,424.029,170.081,33.667,156.346
C09914=1047.167,-11.743,424.044,170.079,33.666,156.346
C09915=1047.161,-11.993,424.058,170.077,33.664,156.345
C09916=1047.155,-12.242,424.072,170.076,33.663,156.345
C09917=1047.148,-12.492,424.086,170.074,33.661,156.345
C09918=1047.143,-12.741,424.101,170.072,33.660,156.345
C09919=1047.136,-12.991,424.115,170.070,33.659,156.345
C09920=1047.130,-13.240,424.129,170.068,33.657,156.344
C09921=1047.124,-13.490,424.144,170.066,33.655,156.344
C09922=1047.118,-13.739,424.157,170.064,33.654,156.344
C09923=1047.111,-13.989,424.172,170.062,33.652,156.344
C09924=1047.106,-14.238,424.186,170.060,33.651,156.344
C09925=1047.099,-14.488,424.201,170.059,33.650,156.343
C09926=1047.092,-14.738,424.215,170.057,33.648,156.343
C09927=1047.087,-14.987,424.229,170.055,33.647,156.343
C09928=1047.080,-15.237,424.243,170.053,33.645,156.343
C09929=1047.074,-15.486,424.257,170.051,33.644,156.343
C09930=1047.067,-15.736,424.271,170.049,33.643,156.342
C09931=1047.062,-15.985,424.285,170.047,33.641,156.342
C09932=1047.055,-16.235,424.299,170.045,33.640,156.342
C09933=1047.048,-16.484,424.313,170.043,33.638,156.342
C09934=1047.042,-16.733,424.328,170.041,33.637,156.342
C09935=1047.035,-16.983,424.341,170.040,33.636,156.341
C09936=1047.030,-17.233,424.355,170.038,33.634,156.341
C09937=1047.023,-17.482,424.369,170.036,33.633,156.341
C09938=1047.017,-17.732,424.383,170.034,33.632,156.341
C09939=1047.010,-17.981,424.398,170.032,33.630,156.341
C09940=1047.004,-18.231,424.411,170.030,33.629,156.340
C09941=1046.998,-18.481,424.425,170.028,33.627,156.340
C09942=1046.991,-18.762,424.441,170.026,33.626,156.340
C09943=1046.984,-19.043,424.457,170.024,33.624,156.340
C09944=1046.976,-19.325,424.473,170.022,33.622,156.340
C09945=1046.970,-19.607,424.488,170.019,33.621,156.339
C09946=1046.963,-19.856,424.502,170.017,33.620,156.339
C09947=1046.957,-20.106,424.516,170.016,33.618,156.339
C09948=1046.950,-20.356,424.530,170.014,33.617,156.339
C09949=1046.944,-20.604,424.544,170.012,33.615,156.339
C09950=1046.938,-20.854,424.558,170.010,33.614,156.338
C09951=1046.932,-21.104,424.571,170.008,33.613,156.338
C09952=1046.926,-21.353,424.586,170.006,33.611,156.338
C09953=1046.919,-21.603,424.599,170.004,33.610,156.338
C09954=1046.913,-21.852,424.613,170.002,33.608,156.338
C09955=1046.907,-22.102,424.627,170.000,33.607,156.337
C09956=1046.900,-22.351,424.640,169.998,33.606,156.337
C09957=1046.894,-22.601,424.655,169.996,33.604,156.337
C09958=1046.888,-22.850,424.668,169.994,33.603,156.337
C09959=1046.882,-23.100,424.682,169.992,33.601,156.337
C09960=1046.876,-23.350,424.696,169.990,33.601,156.337
C09961=1046.869,-23.599,424.710,169.989,33.599,156.336
C09962=1046.862,-23.848,424.723,169.987,33.598,156.336
C09963=1046.857,-24.098,424.737,169.985,33.596,156.336
C09964=1046.851,-24.347,424.751,169.983,33.595,156.336
C09965=1046.844,-24.598,424.765,169.981,33.594,156.336
C09966=1046.838,-24.847,424.778,169.979,33.592,156.335
C09967=1046.831,-25.096,424.792,169.977,33.591,156.335
C09968=1046.826,-25.346,424.806,169.975,33.589,156.335
C09969=1046.819,-25.595,424.820,169.973,33.588,156.335
C09970=1046.813,-25.845,424.833,169.971,33.587,156.335
C09971=1046.807,-26.095,424.847,169.969,33.585,156.335
C09972=1046.801,-26.344,424.860,169.967,33.584,156.334
C09973=1046.794,-26.594,424.874,169.965,33.582,156.334
C09974=1046.789,-26.843,424.888,169.963,33.581,156.334
C09975=1046.782,-27.093,424.901,169.961,33.579,156.334
C09976=1046.776,-27.343,424.915,169.959,33.579,156.334
C09977=1046.769,-27.592,424.928,169.957,33.577,156.333
C09978=1046.763,-27.842,424.942,169.955,33.576,156.333
C09979=1046.757,-28.091,424.955,169.953,33.574,156.333
C09980=1046.751,-28.341,424.969,169.951,33.574,156.333
C09981=1046.744,-28.591,424.982,169.949,33.572,156.333
C09982=1046.738,-28.840,424.996,169.947,33.571,156.333
C09983=1046.732,-29.089,425.009,169.945,33.569,156.332
C09984=1046.725,-29.339,425.023,169.943,33.568,156.332
C09985=1046.719,-29.588,425.036,169.941,33.567,156.332
C09986=1046.713,-29.838,425.050,169.939,33.566,156.332
C09987=1046.706,-30.088,425.063,169.938,33.564,156.332
C09988=1046.700,-30.337,425.077,169.936,33.563,156.332
C09989=1046.694,-30.586,425.090,169.934,33.562,156.332
C09990=1046.687,-30.836,425.104,169.932,33.561,156.331
C09991=1046.681,-31.086,425.117,169.930,33.559,156.331
C09992=1046.675,-31.335,425.130,169.928,33.558,156.331
C09993=1046.668,-31.585,425.144,169.926,33.557,156.331
C09994=1046.662,-31.834,425.157,169.924,33.556,156.331
C09995=1046.655,-32.083,425.170,169.922,33.554,156.330
C09996=1046.650,-32.333,425.184,169.920,33.553,156.330
//INST
///DATE 2021/06/25 14:47
///ATTR SC,RW,RJ
////FRAME ROBOT
///GROUP1 RB1
NOP
MOVL C00000 V=800.0 PL=0
MOVL C00001 V=800.0 PL=0
MOVL C00002 V=800.0 PL=0
MOVL C00003 V=800.0 PL=0
MOVL C00004 V=800.0 PL=0
MOVL C00005 V=800.0 PL=0
MOVL C00006 V=800.0 PL=0
MOVL C00007 V=800.0 PL=0
MOVL C00008 V=800.0 PL=0
MOVL C00009 V=800.0 PL=0
MOVL C00010 V=800.0 PL=0
MOVL C00011 V=800.0 PL=0
MOVL C00012 V=800.0 PL=0
MOVL C00013 V=800.0 PL=0
MOVL C00014 V=800.0 PL=0
MOVL C00015 V=800.0 PL=0
MOVL C00016 V=800.0 PL=0
MOVL C00017 V=800.0 PL=0
MOVL C00018 V=800.0 PL=0
MOVL C00019 V=800.0 PL=0
MOVL C00020 V=800.0 PL=0
MOVL C00021 V=800.0 PL=0
MOVL C00022 V=800.0 PL=0
MOVL C00023 V=800.0 PL=0
MOVL C00024 V=800.0 PL=0
MOVL C00025 V=800.0 PL=0
MOVL C00026 V=800.0 PL=0
MOVL C00027 V=800.0 PL=0
MOVL C00028 V=800.0 PL=0
MOVL C00029 V=800.0 PL=0
MOVL C00030 V=800.0 PL=0
MOVL C00031 V=800.0 PL=0
MOVL C00032 V=800.0 PL=0
MOVL C00033 V=800.0 PL=0
MOVL C00034 V=800.0 PL=0
MOVL C00035 V=800.0 PL=0
MOVL C00036 V=800.0 PL=0
MOVL C00037 V=800.0 PL=0
MOVL C00038 V=800.0 PL=0
MOVL C00039 V=800.0 PL=0
MOVL C00040 V=800.0 PL=0
MOVL C00041 V=800.0 PL=0
MOVL C00042 V=800.0 PL=0
MOVL C00043 V=800.0 PL=0
MOVL C00044 V=800.0 PL=0
MOVL C00045 V=800.0 PL=0
MOVL C00046 V=800.0 PL=0
MOVL C00047 V=800.0 PL=0
MOVL C00048 V=800.0 PL=0
MOVL C00049 V=800.0 PL=0
MOVL C00050 V=800.0 PL=0
MOVL C00051 V=800.0 PL=0
MOVL C00052 V=800.0 PL=0
MOVL C00053 V=800.0 PL=0
MOVL C00054 V=800.0 PL=0
MOVL C00055 V=800.0 PL=0
MOVL C00056 V=800.0 PL=0
MOVL C00057 V=800.0 PL=0
MOVL C00058 V=800.0 PL=0
MOVL C00059 V=800.0 PL=0
MOVL C00060 V=800.0 PL=0
MOVL C00061 V=800.0 PL=0
MOVL C00062 V=800.0 PL=0
MOVL C00063 V=800.0 PL=0
MOVL C00064 V=800.0 PL=0
MOVL C00065 V=800.0 PL=0
MOVL C00066 V=800.0 PL=0
MOVL C00067 V=800.0 PL=0
MOVL C00068 V=800.0 PL=0
MOVL C00069 V=800.0 PL=0
MOVL C00070 V=800.0 PL=0
MOVL C00071 V=800.0 PL=0
MOVL C00072 V=800.0 PL=0
MOVL C00073 V=800.0 PL=0
MOVL C00074 V=800.0 PL=0
MOVL C00075 V=800.0 PL=0
MOVL C00076 V=800.0 PL=0
MOVL C00077 V=800.0 PL=0
MOVL C00078 V=800.0 PL=0
MOVL C00079 V=800.0 PL=0
MOVL C00080 V=800.0 PL=0
MOVL C00081 V=800.0 PL=0
MOVL C00082 V=800.0 PL=0
MOVL C00083 V=800.0 PL=0
MOVL C00084 V=800.0 PL=0
MOVL C00085 V=800.0 PL=0
MOVL C00086 V=800.0 PL=0
MOVL C00087 V=800.0 PL=0
MOVL C00088 V=800.0 PL=0
MOVL C00089 V=800.0 PL=0
MOVL C00090 V=800.0 PL=0
MOVL C00091 V=800.0 PL=0
MOVL C00092 V=800.0 PL=0
MOVL C00093 V=800.0 PL=0
MOVL C00094 V=800.0 PL=0
MOVL C00095 V=800.0 PL=0
MOVL C00096 V=800.0 PL=0
MOVL C00097 V=800.0 PL=0
MOVL C00098 V=800.0 PL=0
MOVL C00099 V=800.0 PL=0
MOVL C00100 V=800.0 PL=0
MOVL C00101 V=800.0 PL=0
MOVL C00102 V=800.0 PL=0
MOVL C00103 V=800.0 PL=0
MOVL C00104 V=800.0 PL=0
MOVL C00105 V=800.0 PL=0
MOVL C00106 V=800.0 PL=0
MOVL C00107 V=800.0 PL=0
MOVL C00108 V=800.0 PL=0
MOVL C00109 V=800.0 PL=0
MOVL C00110 V=800.0 PL=0
MOVL C00111 V=800.0 PL=0
MOVL C00112 V=800.0 PL=0
MOVL C00113 V=800.0 PL=0
MOVL C00114 V=800.0 PL=0
MOVL C00115 V=800.0 PL=0
MOVL C00116 V=800.0 PL=0
MOVL C00117 V=800.0 PL=0
MOVL C00118 V=800.0 PL=0
MOVL C00119 V=800.0 PL=0
MOVL C00120 V=800.0 PL=0
MOVL C00121 V=800.0 PL=0
MOVL C00122 V=800.0 PL=0
MOVL C00123 V=800.0 PL=0
MOVL C00124 V=800.0 PL=0
MOVL C00125 V=800.0 PL=0
MOVL C00126 V=800.0 PL=0
MOVL C00127 V=800.0 PL=0
MOVL C00128 V=800.0 PL=0
MOVL C00129 V=800.0 PL=0
MOVL C00130 V=800.0 PL=0
MOVL C00131 V=800.0 PL=0
MOVL C00132 V=800.0 PL=0
MOVL C00133 V=800.0 PL=0
MOVL C00134 V=800.0 PL=0
MOVL C00135 V=800.0 PL=0
MOVL C00136 V=800.0 PL=0
MOVL C00137 V=800.0 PL=0
MOVL C00138 V=800.0 PL=0
MOVL C00139 V=800.0 PL=0
MOVL C00140 V=800.0 PL=0
MOVL C00141 V=800.0 PL=0
MOVL C00142 V=800.0 PL=0
MOVL C00143 V=800.0 PL=0
MOVL C00144 V=800.0 PL=0
MOVL C00145 V=800.0 PL=0
MOVL C00146 V=800.0 PL=0
MOVL C00147 V=800.0 PL=0
MOVL C00148 V=800.0 PL=0
MOVL C00149 V=800.0 PL=0
MOVL C00150 V=800.0 PL=0
MOVL C00151 V=800.0 PL=0
MOVL C00152 V=800.0 PL=0
MOVL C00153 V=800.0 PL=0
MOVL C00154 V=800.0 PL=0
MOVL C00155 V=800.0 PL=0
MOVL C00156 V=800.0 PL=0
MOVL C00157 V=800.0 PL=0
MOVL C00158 V=800.0 PL=0
MOVL C00159 V=800.0 PL=0
MOVL C00160 V=800.0 PL=0
MOVL C00161 V=800.0 PL=0
MOVL C00162 V=800.0 PL=0
MOVL C00163 V=800.0 PL=0
MOVL C00164 V=800.0 PL=0
MOVL C00165 V=800.0 PL=0
MOVL C00166 V=800.0 PL=0
MOVL C00167 V=800.0 PL=0
MOVL C00168 V=800.0 PL=0
MOVL C00169 V=800.0 PL=0
MOVL C00170 V=800.0 PL=0
MOVL C00171 V=800.0 PL=0
MOVL C00172 V=800.0 PL=0
MOVL C00173 V=800.0 PL=0
MOVL C00174 V=800.0 PL=0
MOVL C00175 V=800.0 PL=0
MOVL C00176 V=800.0 PL=0
MOVL C00177 V=800.0 PL=0
MOVL C00178 V=800.0 PL=0
MOVL C00179 V=800.0 PL=0
MOVL C00180 V=800.0 PL=0
MOVL C00181 V=800.0 PL=0
MOVL C00182 V=800.0 PL=0
MOVL C00183 V=800.0 PL=0
MOVL C00184 V=800.0 PL=0
MOVL C00185 V=800.0 PL=0
MOVL C00186 V=800.0 PL=0
MOVL C00187 V=800.0 PL=0
MOVL C00188 V=800.0 PL=0
MOVL C00189 V=800.0 PL=0
MOVL C00190 V=800.0 PL=0
MOVL C00191 V=800.0 PL=0
MOVL C00192 V=800.0 PL=0
MOVL C00193 V=800.0 PL=0
MOVL C00194 V=800.0 PL=0
MOVL C00195 V=800.0 PL=0
MOVL C00196 V=800.0 PL=0
MOVL C00197 V=800.0 PL=0
MOVL C00198 V=800.0 PL=0
MOVL C00199 V=800.0 PL=0
MOVL C00200 V=800.0 PL=0
MOVL C00201 V=800.0 PL=0
MOVL C00202 V=800.0 PL=0
MOVL C00203 V=800.0 PL=0
MOVL C00204 V=800.0 PL=0
MOVL C00205 V=800.0 PL=0
MOVL C00206 V=800.0 PL=0
MOVL C00207 V=800.0 PL=0
MOVL C00208 V=800.0 PL=0
MOVL C00209 V=800.0 PL=0
MOVL C00210 V=800.0 PL=0
MOVL C00211 V=800.0 PL=0
MOVL C00212 V=800.0 PL=0
MOVL C00213 V=800.0 PL=0
MOVL C00214 V=800.0 PL=0
MOVL C00215 V=800.0 PL=0
MOVL C00216 V=800.0 PL=0
MOVL C00217 V=800.0 PL=0
MOVL C00218 V=800.0 PL=0
MOVL C00219 V=800.0 PL=0
MOVL C00220 V=800.0 PL=0
MOVL C00221 V=800.0 PL=0
MOVL C00222 V=800.0 PL=0
MOVL C00223 V=800.0 PL=0
MOVL C00224 V=800.0 PL=0
MOVL C00225 V=800.0 PL=0
MOVL C00226 V=800.0 PL=0
MOVL C00227 V=800.0 PL=0
MOVL C00228 V=800.0 PL=0
MOVL C00229 V=800.0 PL=0
MOVL C00230 V=800.0 PL=0
MOVL C00231 V=800.0 PL=0
MOVL C00232 V=800.0 PL=0
MOVL C00233 V=800.0 PL=0
MOVL C00234 V=800.0 PL=0
MOVL C00235 V=800.0 PL=0
MOVL C00236 V=800.0 PL=0
MOVL C00237 V=800.0 PL=0
MOVL C00238 V=800.0 PL=0
MOVL C00239 V=800.0 PL=0
MOVL C00240 V=800.0 PL=0
MOVL C00241 V=800.0 PL=0
MOVL C00242 V=800.0 PL=0
MOVL C00243 V=800.0 PL=0
MOVL C00244 V=800.0 PL=0
MOVL C00245 V=800.0 PL=0
MOVL C00246 V=800.0 PL=0
MOVL C00247 V=800.0 PL=0
MOVL C00248 V=800.0 PL=0
MOVL C00249 V=800.0 PL=0
MOVL C00250 V=800.0 PL=0
MOVL C00251 V=800.0 PL=0
MOVL C00252 V=800.0 PL=0
MOVL C00253 V=800.0 PL=0
MOVL C00254 V=800.0 PL=0
MOVL C00255 V=800.0 PL=0
MOVL C00256 V=800.0 PL=0
MOVL C00257 V=800.0 PL=0
MOVL C00258 V=800.0 PL=0
MOVL C00259 V=800.0 PL=0
MOVL C00260 V=800.0 PL=0
MOVL C00261 V=800.0 PL=0
MOVL C00262 V=800.0 PL=0
MOVL C00263 V=800.0 PL=0
MOVL C00264 V=800.0 PL=0
MOVL C00265 V=800.0 PL=0
MOVL C00266 V=800.0 PL=0
MOVL C00267 V=800.0 PL=0
MOVL C00268 V=800.0 PL=0
MOVL C00269 V=800.0 PL=0
MOVL C00270 V=800.0 PL=0
MOVL C00271 V=800.0 PL=0
MOVL C00272 V=800.0 PL=0
MOVL C00273 V=800.0 PL=0
MOVL C00274 V=800.0 PL=0
MOVL C00275 V=800.0 PL=0
MOVL C00276 V=800.0 PL=0
MOVL C00277 V=800.0 PL=0
MOVL C00278 V=800.0 PL=0
MOVL C00279 V=800.0 PL=0
MOVL C00280 V=800.0 PL=0
MOVL C00281 V=800.0 PL=0
MOVL C00282 V=800.0 PL=0
MOVL C00283 V=800.0 PL=0
MOVL C00284 V=800.0 PL=0
MOVL C00285 V=800.0 PL=0
MOVL C00286 V=800.0 PL=0
MOVL C00287 V=800.0 PL=0
MOVL C00288 V=800.0 PL=0
MOVL C00289 V=800.0 PL=0
MOVL C00290 V=800.0 PL=0
MOVL C00291 V=800.0 PL=0
MOVL C00292 V=800.0 PL=0
MOVL C00293 V=800.0 PL=0
MOVL C00294 V=800.0 PL=0
MOVL C00295 V=800.0 PL=0
MOVL C00296 V=800.0 PL=0
MOVL C00297 V=800.0 PL=0
MOVL C00298 V=800.0 PL=0
MOVL C00299 V=800.0 PL=0
MOVL C00300 V=800.0 PL=0
MOVL C00301 V=800.0 PL=0
MOVL C00302 V=800.0 PL=0
MOVL C00303 V=800.0 PL=0
MOVL C00304 V=800.0 PL=0
MOVL C00305 V=800.0 PL=0
MOVL C00306 V=800.0 PL=0
MOVL C00307 V=800.0 PL=0
MOVL C00308 V=800.0 PL=0
MOVL C00309 V=800.0 PL=0
MOVL C00310 V=800.0 PL=0
MOVL C00311 V=800.0 PL=0
MOVL C00312 V=800.0 PL=0
MOVL C00313 V=800.0 PL=0
MOVL C00314 V=800.0 PL=0
MOVL C00315 V=800.0 PL=0
MOVL C00316 V=800.0 PL=0
MOVL C00317 V=800.0 PL=0
MOVL C00318 V=800.0 PL=0
MOVL C00319 V=800.0 PL=0
MOVL C00320 V=800.0 PL=0
MOVL C00321 V=800.0 PL=0
MOVL C00322 V=800.0 PL=0
MOVL C00323 V=800.0 PL=0
MOVL C00324 V=800.0 PL=0
MOVL C00325 V=800.0 PL=0
MOVL C00326 V=800.0 PL=0
MOVL C00327 V=800.0 PL=0
MOVL C00328 V=800.0 PL=0
MOVL C00329 V=800.0 PL=0
MOVL C00330 V=800.0 PL=0
MOVL C00331 V=800.0 PL=0
MOVL C00332 V=800.0 PL=0
MOVL C00333 V=800.0 PL=0
MOVL C00334 V=800.0 PL=0
MOVL C00335 V=800.0 PL=0
MOVL C00336 V=800.0 PL=0
MOVL C00337 V=800.0 PL=0
MOVL C00338 V=800.0 PL=0
MOVL C00339 V=800.0 PL=0
MOVL C00340 V=800.0 PL=0
MOVL C00341 V=800.0 PL=0
MOVL C00342 V=800.0 PL=0
MOVL C00343 V=800.0 PL=0
MOVL C00344 V=800.0 PL=0
MOVL C00345 V=800.0 PL=0
MOVL C00346 V=800.0 PL=0
MOVL C00347 V=800.0 PL=0
MOVL C00348 V=800.0 PL=0
MOVL C00349 V=800.0 PL=0
MOVL C00350 V=800.0 PL=0
MOVL C00351 V=800.0 PL=0
MOVL C00352 V=800.0 PL=0
MOVL C00353 V=800.0 PL=0
MOVL C00354 V=800.0 PL=0
MOVL C00355 V=800.0 PL=0
MOVL C00356 V=800.0 PL=0
MOVL C00357 V=800.0 PL=0
MOVL C00358 V=800.0 PL=0
MOVL C00359 V=800.0 PL=0
MOVL C00360 V=800.0 PL=0
MOVL C00361 V=800.0 PL=0
MOVL C00362 V=800.0 PL=0
MOVL C00363 V=800.0 PL=0
MOVL C00364 V=800.0 PL=0
MOVL C00365 V=800.0 PL=0
MOVL C00366 V=800.0 PL=0
MOVL C00367 V=800.0 PL=0
MOVL C00368 V=800.0 PL=0
MOVL C00369 V=800.0 PL=0
MOVL C00370 V=800.0 PL=0
MOVL C00371 V=800.0 PL=0
MOVL C00372 V=800.0 PL=0
MOVL C00373 V=800.0 PL=0
MOVL C00374 V=800.0 PL=0
MOVL C00375 V=800.0 PL=0
MOVL C00376 V=800.0 PL=0
MOVL C00377 V=800.0 PL=0
MOVL C00378 V=800.0 PL=0
MOVL C00379 V=800.0 PL=0
MOVL C00380 V=800.0 PL=0
MOVL C00381 V=800.0 PL=0
MOVL C00382 V=800.0 PL=0
MOVL C00383 V=800.0 PL=0
MOVL C00384 V=800.0 PL=0
MOVL C00385 V=800.0 PL=0
MOVL C00386 V=800.0 PL=0
MOVL C00387 V=800.0 PL=0
MOVL C00388 V=800.0 PL=0
MOVL C00389 V=800.0 PL=0
MOVL C00390 V=800.0 PL=0
MOVL C00391 V=800.0 PL=0
MOVL C00392 V=800.0 PL=0
MOVL C00393 V=800.0 PL=0
MOVL C00394 V=800.0 PL=0
MOVL C00395 V=800.0 PL=0
MOVL C00396 V=800.0 PL=0
MOVL C00397 V=800.0 PL=0
MOVL C00398 V=800.0 PL=0
MOVL C00399 V=800.0 PL=0
MOVL C00400 V=800.0 PL=0
MOVL C00401 V=800.0 PL=0
MOVL C00402 V=800.0 PL=0
MOVL C00403 V=800.0 PL=0
MOVL C00404 V=800.0 PL=0
MOVL C00405 V=800.0 PL=0
MOVL C00406 V=800.0 PL=0
MOVL C00407 V=800.0 PL=0
MOVL C00408 V=800.0 PL=0
MOVL C00409 V=800.0 PL=0
MOVL C00410 V=800.0 PL=0
MOVL C00411 V=800.0 PL=0
MOVL C00412 V=800.0 PL=0
MOVL C00413 V=800.0 PL=0
MOVL C00414 V=800.0 PL=0
MOVL C00415 V=800.0 PL=0
MOVL C00416 V=800.0 PL=0
MOVL C00417 V=800.0 PL=0
MOVL C00418 V=800.0 PL=0
MOVL C00419 V=800.0 PL=0
MOVL C00420 V=800.0 PL=0
MOVL C00421 V=800.0 PL=0
MOVL C00422 V=800.0 PL=0
MOVL C00423 V=800.0 PL=0
MOVL C00424 V=800.0 PL=0
MOVL C00425 V=800.0 PL=0
MOVL C00426 V=800.0 PL=0
MOVL C00427 V=800.0 PL=0
MOVL C00428 V=800.0 PL=0
MOVL C00429 V=800.0 PL=0
MOVL C00430 V=800.0 PL=0
MOVL C00431 V=800.0 PL=0
MOVL C00432 V=800.0 PL=0
MOVL C00433 V=800.0 PL=0
MOVL C00434 V=800.0 PL=0
MOVL C00435 V=800.0 PL=0
MOVL C00436 V=800.0 PL=0
MOVL C00437 V=800.0 PL=0
MOVL C00438 V=800.0 PL=0
MOVL C00439 V=800.0 PL=0
MOVL C00440 V=800.0 PL=0
MOVL C00441 V=800.0 PL=0
MOVL C00442 V=800.0 PL=0
MOVL C00443 V=800.0 PL=0
MOVL C00444 V=800.0 PL=0
MOVL C00445 V=800.0 PL=0
MOVL C00446 V=800.0 PL=0
MOVL C00447 V=800.0 PL=0
MOVL C00448 V=800.0 PL=0
MOVL C00449 V=800.0 PL=0
MOVL C00450 V=800.0 PL=0
MOVL C00451 V=800.0 PL=0
MOVL C00452 V=800.0 PL=0
MOVL C00453 V=800.0 PL=0
MOVL C00454 V=800.0 PL=0
MOVL C00455 V=800.0 PL=0
MOVL C00456 V=800.0 PL=0
MOVL C00457 V=800.0 PL=0
MOVL C00458 V=800.0 PL=0
MOVL C00459 V=800.0 PL=0
MOVL C00460 V=800.0 PL=0
MOVL C00461 V=800.0 PL=0
MOVL C00462 V=800.0 PL=0
MOVL C00463 V=800.0 PL=0
MOVL C00464 V=800.0 PL=0
MOVL C00465 V=800.0 PL=0
MOVL C00466 V=800.0 PL=0
MOVL C00467 V=800.0 PL=0
MOVL C00468 V=800.0 PL=0
MOVL C00469 V=800.0 PL=0
MOVL C00470 V=800.0 PL=0
MOVL C00471 V=800.0 PL=0
MOVL C00472 V=800.0 PL=0
MOVL C00473 V=800.0 PL=0
MOVL C00474 V=800.0 PL=0
MOVL C00475 V=800.0 PL=0
MOVL C00476 V=800.0 PL=0
MOVL C00477 V=800.0 PL=0
MOVL C00478 V=800.0 PL=0
MOVL C00479 V=800.0 PL=0
MOVL C00480 V=800.0 PL=0
MOVL C00481 V=800.0 PL=0
MOVL C00482 V=800.0 PL=0
MOVL C00483 V=800.0 PL=0
MOVL C00484 V=800.0 PL=0
MOVL C00485 V=800.0 PL=0
MOVL C00486 V=800.0 PL=0
MOVL C00487 V=800.0 PL=0
MOVL C00488 V=800.0 PL=0
MOVL C00489 V=800.0 PL=0
MOVL C00490 V=800.0 PL=0
MOVL C00491 V=800.0 PL=0
MOVL C00492 V=800.0 PL=0
MOVL C00493 V=800.0 PL=0
MOVL C00494 V=800.0 PL=0
MOVL C00495 V=800.0 PL=0
MOVL C00496 V=800.0 PL=0
MOVL C00497 V=800.0 PL=0
MOVL C00498 V=800.0 PL=0
MOVL C00499 V=800.0 PL=0
MOVL C00500 V=800.0 PL=0
MOVL C00501 V=800.0 PL=0
MOVL C00502 V=800.0 PL=0
MOVL C00503 V=800.0 PL=0
MOVL C00504 V=800.0 PL=0
MOVL C00505 V=800.0 PL=0
MOVL C00506 V=800.0 PL=0
MOVL C00507 V=800.0 PL=0
MOVL C00508 V=800.0 PL=0
MOVL C00509 V=800.0 PL=0
MOVL C00510 V=800.0 PL=0
MOVL C00511 V=800.0 PL=0
MOVL C00512 V=800.0 PL=0
MOVL C00513 V=800.0 PL=0
MOVL C00514 V=800.0 PL=0
MOVL C00515 V=800.0 PL=0
MOVL C00516 V=800.0 PL=0
MOVL C00517 V=800.0 PL=0
MOVL C00518 V=800.0 PL=0
MOVL C00519 V=800.0 PL=0
MOVL C00520 V=800.0 PL=0
MOVL C00521 V=800.0 PL=0
MOVL C00522 V=800.0 PL=0
MOVL C00523 V=800.0 PL=0
MOVL C00524 V=800.0 PL=0
MOVL C00525 V=800.0 PL=0
MOVL C00526 V=800.0 PL=0
MOVL C00527 V=800.0 PL=0
MOVL C00528 V=800.0 PL=0
MOVL C00529 V=800.0 PL=0
MOVL C00530 V=800.0 PL=0
MOVL C00531 V=800.0 PL=0
MOVL C00532 V=800.0 PL=0
MOVL C00533 V=800.0 PL=0
MOVL C00534 V=800.0 PL=0
MOVL C00535 V=800.0 PL=0
MOVL C00536 V=800.0 PL=0
MOVL C00537 V=800.0 PL=0
MOVL C00538 V=800.0 PL=0
MOVL C00539 V=800.0 PL=0
MOVL C00540 V=800.0 PL=0
MOVL C00541 V=800.0 PL=0
MOVL C00542 V=800.0 PL=0
MOVL C00543 V=800.0 PL=0
MOVL C00544 V=800.0 PL=0
MOVL C00545 V=800.0 PL=0
MOVL C00546 V=800.0 PL=0
MOVL C00547 V=800.0 PL=0
MOVL C00548 V=800.0 PL=0
MOVL C00549 V=800.0 PL=0
MOVL C00550 V=800.0 PL=0
MOVL C00551 V=800.0 PL=0
MOVL C00552 V=800.0 PL=0
MOVL C00553 V=800.0 PL=0
MOVL C00554 V=800.0 PL=0
MOVL C00555 V=800.0 PL=0
MOVL C00556 V=800.0 PL=0
MOVL C00557 V=800.0 PL=0
MOVL C00558 V=800.0 PL=0
MOVL C00559 V=800.0 PL=0
MOVL C00560 V=800.0 PL=0
MOVL C00561 V=800.0 PL=0
MOVL C00562 V=800.0 PL=0
MOVL C00563 V=800.0 PL=0
MOVL C00564 V=800.0 PL=0
MOVL C00565 V=800.0 PL=0
MOVL C00566 V=800.0 PL=0
MOVL C00567 V=800.0 PL=0
MOVL C00568 V=800.0 PL=0
MOVL C00569 V=800.0 PL=0
MOVL C00570 V=800.0 PL=0
MOVL C00571 V=800.0 PL=0
MOVL C00572 V=800.0 PL=0
MOVL C00573 V=800.0 PL=0
MOVL C00574 V=800.0 PL=0
MOVL C00575 V=800.0 PL=0
MOVL C00576 V=800.0 PL=0
MOVL C00577 V=800.0 PL=0
MOVL C00578 V=800.0 PL=0
MOVL C00579 V=800.0 PL=0
MOVL C00580 V=800.0 PL=0
MOVL C00581 V=800.0 PL=0
MOVL C00582 V=800.0 PL=0
MOVL C00583 V=800.0 PL=0
MOVL C00584 V=800.0 PL=0
MOVL C00585 V=800.0 PL=0
MOVL C00586 V=800.0 PL=0
MOVL C00587 V=800.0 PL=0
MOVL C00588 V=800.0 PL=0
MOVL C00589 V=800.0 PL=0
MOVL C00590 V=800.0 PL=0
MOVL C00591 V=800.0 PL=0
MOVL C00592 V=800.0 PL=0
MOVL C00593 V=800.0 PL=0
MOVL C00594 V=800.0 PL=0
MOVL C00595 V=800.0 PL=0
MOVL C00596 V=800.0 PL=0
MOVL C00597 V=800.0 PL=0
MOVL C00598 V=800.0 PL=0
MOVL C00599 V=800.0 PL=0
MOVL C00600 V=800.0 PL=0
MOVL C00601 V=800.0 PL=0
MOVL C00602 V=800.0 PL=0
MOVL C00603 V=800.0 PL=0
MOVL C00604 V=800.0 PL=0
MOVL C00605 V=800.0 PL=0
MOVL C00606 V=800.0 PL=0
MOVL C00607 V=800.0 PL=0
MOVL C00608 V=800.0 PL=0
MOVL C00609 V=800.0 PL=0
MOVL C00610 V=800.0 PL=0
MOVL C00611 V=800.0 PL=0
MOVL C00612 V=800.0 PL=0
MOVL C00613 V=800.0 PL=0
MOVL C00614 V=800.0 PL=0
MOVL C00615 V=800.0 PL=0
MOVL C00616 V=800.0 PL=0
MOVL C00617 V=800.0 PL=0
MOVL C00618 V=800.0 PL=0
MOVL C00619 V=800.0 PL=0
MOVL C00620 V=800.0 PL=0
MOVL C00621 V=800.0 PL=0
MOVL C00622 V=800.0 PL=0
MOVL C00623 V=800.0 PL=0
MOVL C00624 V=800.0 PL=0
MOVL C00625 V=800.0 PL=0
MOVL C00626 V=800.0 PL=0
MOVL C00627 V=800.0 PL=0
MOVL C00628 V=800.0 PL=0
MOVL C00629 V=800.0 PL=0
MOVL C00630 V=800.0 PL=0
MOVL C00631 V=800.0 PL=0
MOVL C00632 V=800.0 PL=0
MOVL C00633 V=800.0 PL=0
MOVL C00634 V=800.0 PL=0
MOVL C00635 V=800.0 PL=0
MOVL C00636 V=800.0 PL=0
MOVL C00637 V=800.0 PL=0
MOVL C00638 V=800.0 PL=0
MOVL C00639 V=800.0 PL=0
MOVL C00640 V=800.0 PL=0
MOVL C00641 V=800.0 PL=0
MOVL C00642 V=800.0 PL=0
MOVL C00643 V=800.0 PL=0
MOVL C00644 V=800.0 PL=0
MOVL C00645 V=800.0 PL=0
MOVL C00646 V=800.0 PL=0
MOVL C00647 V=800.0 PL=0
MOVL C00648 V=800.0 PL=0
MOVL C00649 V=800.0 PL=0
MOVL C00650 V=800.0 PL=0
MOVL C00651 V=800.0 PL=0
MOVL C00652 V=800.0 PL=0
MOVL C00653 V=800.0 PL=0
MOVL C00654 V=800.0 PL=0
MOVL C00655 V=800.0 PL=0
MOVL C00656 V=800.0 PL=0
MOVL C00657 V=800.0 PL=0
MOVL C00658 V=800.0 PL=0
MOVL C00659 V=800.0 PL=0
MOVL C00660 V=800.0 PL=0
MOVL C00661 V=800.0 PL=0
MOVL C00662 V=800.0 PL=0
MOVL C00663 V=800.0 PL=0
MOVL C00664 V=800.0 PL=0
MOVL C00665 V=800.0 PL=0
MOVL C00666 V=800.0 PL=0
MOVL C00667 V=800.0 PL=0
MOVL C00668 V=800.0 PL=0
MOVL C00669 V=800.0 PL=0
MOVL C00670 V=800.0 PL=0
MOVL C00671 V=800.0 PL=0
MOVL C00672 V=800.0 PL=0
MOVL C00673 V=800.0 PL=0
MOVL C00674 V=800.0 PL=0
MOVL C00675 V=800.0 PL=0
MOVL C00676 V=800.0 PL=0
MOVL C00677 V=800.0 PL=0
MOVL C00678 V=800.0 PL=0
MOVL C00679 V=800.0 PL=0
MOVL C00680 V=800.0 PL=0
MOVL C00681 V=800.0 PL=0
MOVL C00682 V=800.0 PL=0
MOVL C00683 V=800.0 PL=0
MOVL C00684 V=800.0 PL=0
MOVL C00685 V=800.0 PL=0
MOVL C00686 V=800.0 PL=0
MOVL C00687 V=800.0 PL=0
MOVL C00688 V=800.0 PL=0
MOVL C00689 V=800.0 PL=0
MOVL C00690 V=800.0 PL=0
MOVL C00691 V=800.0 PL=0
MOVL C00692 V=800.0 PL=0
MOVL C00693 V=800.0 PL=0
MOVL C00694 V=800.0 PL=0
MOVL C00695 V=800.0 PL=0
MOVL C00696 V=800.0 PL=0
MOVL C00697 V=800.0 PL=0
MOVL C00698 V=800.0 PL=0
MOVL C00699 V=800.0 PL=0
MOVL C00700 V=800.0 PL=0
MOVL C00701 V=800.0 PL=0
MOVL C00702 V=800.0 PL=0
MOVL C00703 V=800.0 PL=0
MOVL C00704 V=800.0 PL=0
MOVL C00705 V=800.0 PL=0
MOVL C00706 V=800.0 PL=0
MOVL C00707 V=800.0 PL=0
MOVL C00708 V=800.0 PL=0
MOVL C00709 V=800.0 PL=0
MOVL C00710 V=800.0 PL=0
MOVL C00711 V=800.0 PL=0
MOVL C00712 V=800.0 PL=0
MOVL C00713 V=800.0 PL=0
MOVL C00714 V=800.0 PL=0
MOVL C00715 V=800.0 PL=0
MOVL C00716 V=800.0 PL=0
MOVL C00717 V=800.0 PL=0
MOVL C00718 V=800.0 PL=0
MOVL C00719 V=800.0 PL=0
MOVL C00720 V=800.0 PL=0
MOVL C00721 V=800.0 PL=0
MOVL C00722 V=800.0 PL=0
MOVL C00723 V=800.0 PL=0
MOVL C00724 V=800.0 PL=0
MOVL C00725 V=800.0 PL=0
MOVL C00726 V=800.0 PL=0
MOVL C00727 V=800.0 PL=0
MOVL C00728 V=800.0 PL=0
MOVL C00729 V=800.0 PL=0
MOVL C00730 V=800.0 PL=0
MOVL C00731 V=800.0 PL=0
MOVL C00732 V=800.0 PL=0
MOVL C00733 V=800.0 PL=0
MOVL C00734 V=800.0 PL=0
MOVL C00735 V=800.0 PL=0
MOVL C00736 V=800.0 PL=0
MOVL C00737 V=800.0 PL=0
MOVL C00738 V=800.0 PL=0
MOVL C00739 V=800.0 PL=0
MOVL C00740 V=800.0 PL=0
MOVL C00741 V=800.0 PL=0
MOVL C00742 V=800.0 PL=0
MOVL C00743 V=800.0 PL=0
MOVL C00744 V=800.0 PL=0
MOVL C00745 V=800.0 PL=0
MOVL C00746 V=800.0 PL=0
MOVL C00747 V=800.0 PL=0
MOVL C00748 V=800.0 PL=0
MOVL C00749 V=800.0 PL=0
MOVL C00750 V=800.0 PL=0
MOVL C00751 V=800.0 PL=0
MOVL C00752 V=800.0 PL=0
MOVL C00753 V=800.0 PL=0
MOVL C00754 V=800.0 PL=0
MOVL C00755 V=800.0 PL=0
MOVL C00756 V=800.0 PL=0
MOVL C00757 V=800.0 PL=0
MOVL C00758 V=800.0 PL=0
MOVL C00759 V=800.0 PL=0
MOVL C00760 V=800.0 PL=0
MOVL C00761 V=800.0 PL=0
MOVL C00762 V=800.0 PL=0
MOVL C00763 V=800.0 PL=0
MOVL C00764 V=800.0 PL=0
MOVL C00765 V=800.0 PL=0
MOVL C00766 V=800.0 PL=0
MOVL C00767 V=800.0 PL=0
MOVL C00768 V=800.0 PL=0
MOVL C00769 V=800.0 PL=0
MOVL C00770 V=800.0 PL=0
MOVL C00771 V=800.0 PL=0
MOVL C00772 V=800.0 PL=0
MOVL C00773 V=800.0 PL=0
MOVL C00774 V=800.0 PL=0
MOVL C00775 V=800.0 PL=0
MOVL C00776 V=800.0 PL=0
MOVL C00777 V=800.0 PL=0
MOVL C00778 V=800.0 PL=0
MOVL C00779 V=800.0 PL=0
MOVL C00780 V=800.0 PL=0
MOVL C00781 V=800.0 PL=0
MOVL C00782 V=800.0 PL=0
MOVL C00783 V=800.0 PL=0
MOVL C00784 V=800.0 PL=0
MOVL C00785 V=800.0 PL=0
MOVL C00786 V=800.0 PL=0
MOVL C00787 V=800.0 PL=0
MOVL C00788 V=800.0 PL=0
MOVL C00789 V=800.0 PL=0
MOVL C00790 V=800.0 PL=0
MOVL C00791 V=800.0 PL=0
MOVL C00792 V=800.0 PL=0
MOVL C00793 V=800.0 PL=0
MOVL C00794 V=800.0 PL=0
MOVL C00795 V=800.0 PL=0
MOVL C00796 V=800.0 PL=0
MOVL C00797 V=800.0 PL=0
MOVL C00798 V=800.0 PL=0
MOVL C00799 V=800.0 PL=0
MOVL C00800 V=800.0 PL=0
MOVL C00801 V=800.0 PL=0
MOVL C00802 V=800.0 PL=0
MOVL C00803 V=800.0 PL=0
MOVL C00804 V=800.0 PL=0
MOVL C00805 V=800.0 PL=0
MOVL C00806 V=800.0 PL=0
MOVL C00807 V=800.0 PL=0
MOVL C00808 V=800.0 PL=0
MOVL C00809 V=800.0 PL=0
MOVL C00810 V=800.0 PL=0
MOVL C00811 V=800.0 PL=0
MOVL C00812 V=800.0 PL=0
MOVL C00813 V=800.0 PL=0
MOVL C00814 V=800.0 PL=0
MOVL C00815 V=800.0 PL=0
MOVL C00816 V=800.0 PL=0
MOVL C00817 V=800.0 PL=0
MOVL C00818 V=800.0 PL=0
MOVL C00819 V=800.0 PL=0
MOVL C00820 V=800.0 PL=0
MOVL C00821 V=800.0 PL=0
MOVL C00822 V=800.0 PL=0
MOVL C00823 V=800.0 PL=0
MOVL C00824 V=800.0 PL=0
MOVL C00825 V=800.0 PL=0
MOVL C00826 V=800.0 PL=0
MOVL C00827 V=800.0 PL=0
MOVL C00828 V=800.0 PL=0
MOVL C00829 V=800.0 PL=0
MOVL C00830 V=800.0 PL=0
MOVL C00831 V=800.0 PL=0
MOVL C00832 V=800.0 PL=0
MOVL C00833 V=800.0 PL=0
MOVL C00834 V=800.0 PL=0
MOVL C00835 V=800.0 PL=0
MOVL C00836 V=800.0 PL=0
MOVL C00837 V=800.0 PL=0
MOVL C00838 V=800.0 PL=0
MOVL C00839 V=800.0 PL=0
MOVL C00840 V=800.0 PL=0
MOVL C00841 V=800.0 PL=0
MOVL C00842 V=800.0 PL=0
MOVL C00843 V=800.0 PL=0
MOVL C00844 V=800.0 PL=0
MOVL C00845 V=800.0 PL=0
MOVL C00846 V=800.0 PL=0
MOVL C00847 V=800.0 PL=0
MOVL C00848 V=800.0 PL=0
MOVL C00849 V=800.0 PL=0
MOVL C00850 V=800.0 PL=0
MOVL C00851 V=800.0 PL=0
MOVL C00852 V=800.0 PL=0
MOVL C00853 V=800.0 PL=0
MOVL C00854 V=800.0 PL=0
MOVL C00855 V=800.0 PL=0
MOVL C00856 V=800.0 PL=0
MOVL C00857 V=800.0 PL=0
MOVL C00858 V=800.0 PL=0
MOVL C00859 V=800.0 PL=0
MOVL C00860 V=800.0 PL=0
MOVL C00861 V=800.0 PL=0
MOVL C00862 V=800.0 PL=0
MOVL C00863 V=800.0 PL=0
MOVL C00864 V=800.0 PL=0
MOVL C00865 V=800.0 PL=0
MOVL C00866 V=800.0 PL=0
MOVL C00867 V=800.0 PL=0
MOVL C00868 V=800.0 PL=0
MOVL C00869 V=800.0 PL=0
MOVL C00870 V=800.0 PL=0
MOVL C00871 V=800.0 PL=0
MOVL C00872 V=800.0 PL=0
MOVL C00873 V=800.0 PL=0
MOVL C00874 V=800.0 PL=0
MOVL C00875 V=800.0 PL=0
MOVL C00876 V=800.0 PL=0
MOVL C00877 V=800.0 PL=0
MOVL C00878 V=800.0 PL=0
MOVL C00879 V=800.0 PL=0
MOVL C00880 V=800.0 PL=0
MOVL C00881 V=800.0 PL=0
MOVL C00882 V=800.0 PL=0
MOVL C00883 V=800.0 PL=0
MOVL C00884 V=800.0 PL=0
MOVL C00885 V=800.0 PL=0
MOVL C00886 V=800.0 PL=0
MOVL C00887 V=800.0 PL=0
MOVL C00888 V=800.0 PL=0
MOVL C00889 V=800.0 PL=0
MOVL C00890 V=800.0 PL=0
MOVL C00891 V=800.0 PL=0
MOVL C00892 V=800.0 PL=0
MOVL C00893 V=800.0 PL=0
MOVL C00894 V=800.0 PL=0
MOVL C00895 V=800.0 PL=0
MOVL C00896 V=800.0 PL=0
MOVL C00897 V=800.0 PL=0
MOVL C00898 V=800.0 PL=0
MOVL C00899 V=800.0 PL=0
MOVL C00900 V=800.0 PL=0
MOVL C00901 V=800.0 PL=0
MOVL C00902 V=800.0 PL=0
MOVL C00903 V=800.0 PL=0
MOVL C00904 V=800.0 PL=0
MOVL C00905 V=800.0 PL=0
MOVL C00906 V=800.0 PL=0
MOVL C00907 V=800.0 PL=0
MOVL C00908 V=800.0 PL=0
MOVL C00909 V=800.0 PL=0
MOVL C00910 V=800.0 PL=0
MOVL C00911 V=800.0 PL=0
MOVL C00912 V=800.0 PL=0
MOVL C00913 V=800.0 PL=0
MOVL C00914 V=800.0 PL=0
MOVL C00915 V=800.0 PL=0
MOVL C00916 V=800.0 PL=0
MOVL C00917 V=800.0 PL=0
MOVL C00918 V=800.0 PL=0
MOVL C00919 V=800.0 PL=0
MOVL C00920 V=800.0 PL=0
MOVL C00921 V=800.0 PL=0
MOVL C00922 V=800.0 PL=0
MOVL C00923 V=800.0 PL=0
MOVL C00924 V=800.0 PL=0
MOVL C00925 V=800.0 PL=0
MOVL C00926 V=800.0 PL=0
MOVL C00927 V=800.0 PL=0
MOVL C00928 V=800.0 PL=0
MOVL C00929 V=800.0 PL=0
MOVL C00930 V=800.0 PL=0
MOVL C00931 V=800.0 PL=0
MOVL C00932 V=800.0 PL=0
MOVL C00933 V=800.0 PL=0
MOVL C00934 V=800.0 PL=0
MOVL C00935 V=800.0 PL=0
MOVL C00936 V=800.0 PL=0
MOVL C00937 V=800.0 PL=0
MOVL C00938 V=800.0 PL=0
MOVL C00939 V=800.0 PL=0
MOVL C00940 V=800.0 PL=0
MOVL C00941 V=800.0 PL=0
MOVL C00942 V=800.0 PL=0
MOVL C00943 V=800.0 PL=0
MOVL C00944 V=800.0 PL=0
MOVL C00945 V=800.0 PL=0
MOVL C00946 V=800.0 PL=0
MOVL C00947 V=800.0 PL=0
MOVL C00948 V=800.0 PL=0
MOVL C00949 V=800.0 PL=0
MOVL C00950 V=800.0 PL=0
MOVL C00951 V=800.0 PL=0
MOVL C00952 V=800.0 PL=0
MOVL C00953 V=800.0 PL=0
MOVL C00954 V=800.0 PL=0
MOVL C00955 V=800.0 PL=0
MOVL C00956 V=800.0 PL=0
MOVL C00957 V=800.0 PL=0
MOVL C00958 V=800.0 PL=0
MOVL C00959 V=800.0 PL=0
MOVL C00960 V=800.0 PL=0
MOVL C00961 V=800.0 PL=0
MOVL C00962 V=800.0 PL=0
MOVL C00963 V=800.0 PL=0
MOVL C00964 V=800.0 PL=0
MOVL C00965 V=800.0 PL=0
MOVL C00966 V=800.0 PL=0
MOVL C00967 V=800.0 PL=0
MOVL C00968 V=800.0 PL=0
MOVL C00969 V=800.0 PL=0
MOVL C00970 V=800.0 PL=0
MOVL C00971 V=800.0 PL=0
MOVL C00972 V=800.0 PL=0
MOVL C00973 V=800.0 PL=0
MOVL C00974 V=800.0 PL=0
MOVL C00975 V=800.0 PL=0
MOVL C00976 V=800.0 PL=0
MOVL C00977 V=800.0 PL=0
MOVL C00978 V=800.0 PL=0
MOVL C00979 V=800.0 PL=0
MOVL C00980 V=800.0 PL=0
MOVL C00981 V=800.0 PL=0
MOVL C00982 V=800.0 PL=0
MOVL C00983 V=800.0 PL=0
MOVL C00984 V=800.0 PL=0
MOVL C00985 V=800.0 PL=0
MOVL C00986 V=800.0 PL=0
MOVL C00987 V=800.0 PL=0
MOVL C00988 V=800.0 PL=0
MOVL C00989 V=800.0 PL=0
MOVL C00990 V=800.0 PL=0
MOVL C00991 V=800.0 PL=0
MOVL C00992 V=800.0 PL=0
MOVL C00993 V=800.0 PL=0
MOVL C00994 V=800.0 PL=0
MOVL C00995 V=800.0 PL=0
MOVL C00996 V=800.0 PL=0
MOVL C00997 V=800.0 PL=0
MOVL C00998 V=800.0 PL=0
MOVL C00999 V=800.0 PL=0
MOVL C01000 V=800.0 PL=0
MOVL C01001 V=800.0 PL=0
MOVL C01002 V=800.0 PL=0
MOVL C01003 V=800.0 PL=0
MOVL C01004 V=800.0 PL=0
MOVL C01005 V=800.0 PL=0
MOVL C01006 V=800.0 PL=0
MOVL C01007 V=800.0 PL=0
MOVL C01008 V=800.0 PL=0
MOVL C01009 V=800.0 PL=0
MOVL C01010 V=800.0 PL=0
MOVL C01011 V=800.0 PL=0
MOVL C01012 V=800.0 PL=0
MOVL C01013 V=800.0 PL=0
MOVL C01014 V=800.0 PL=0
MOVL C01015 V=800.0 PL=0
MOVL C01016 V=800.0 PL=0
MOVL C01017 V=800.0 PL=0
MOVL C01018 V=800.0 PL=0
MOVL C01019 V=800.0 PL=0
MOVL C01020 V=800.0 PL=0
MOVL C01021 V=800.0 PL=0
MOVL C01022 V=800.0 PL=0
MOVL C01023 V=800.0 PL=0
MOVL C01024 V=800.0 PL=0
MOVL C01025 V=800.0 PL=0
MOVL C01026 V=800.0 PL=0
MOVL C01027 V=800.0 PL=0
MOVL C01028 V=800.0 PL=0
MOVL C01029 V=800.0 PL=0
MOVL C01030 V=800.0 PL=0
MOVL C01031 V=800.0 PL=0
MOVL C01032 V=800.0 PL=0
MOVL C01033 V=800.0 PL=0
MOVL C01034 V=800.0 PL=0
MOVL C01035 V=800.0 PL=0
MOVL C01036 V=800.0 PL=0
MOVL C01037 V=800.0 PL=0
MOVL C01038 V=800.0 PL=0
MOVL C01039 V=800.0 PL=0
MOVL C01040 V=800.0 PL=0
MOVL C01041 V=800.0 PL=0
MOVL C01042 V=800.0 PL=0
MOVL C01043 V=800.0 PL=0
MOVL C01044 V=800.0 PL=0
MOVL C01045 V=800.0 PL=0
MOVL C01046 V=800.0 PL=0
MOVL C01047 V=800.0 PL=0
MOVL C01048 V=800.0 PL=0
MOVL C01049 V=800.0 PL=0
MOVL C01050 V=800.0 PL=0
MOVL C01051 V=800.0 PL=0
MOVL C01052 V=800.0 PL=0
MOVL C01053 V=800.0 PL=0
MOVL C01054 V=800.0 PL=0
MOVL C01055 V=800.0 PL=0
MOVL C01056 V=800.0 PL=0
MOVL C01057 V=800.0 PL=0
MOVL C01058 V=800.0 PL=0
MOVL C01059 V=800.0 PL=0
MOVL C01060 V=800.0 PL=0
MOVL C01061 V=800.0 PL=0
MOVL C01062 V=800.0 PL=0
MOVL C01063 V=800.0 PL=0
MOVL C01064 V=800.0 PL=0
MOVL C01065 V=800.0 PL=0
MOVL C01066 V=800.0 PL=0
MOVL C01067 V=800.0 PL=0
MOVL C01068 V=800.0 PL=0
MOVL C01069 V=800.0 PL=0
MOVL C01070 V=800.0 PL=0
MOVL C01071 V=800.0 PL=0
MOVL C01072 V=800.0 PL=0
MOVL C01073 V=800.0 PL=0
MOVL C01074 V=800.0 PL=0
MOVL C01075 V=800.0 PL=0
MOVL C01076 V=800.0 PL=0
MOVL C01077 V=800.0 PL=0
MOVL C01078 V=800.0 PL=0
MOVL C01079 V=800.0 PL=0
MOVL C01080 V=800.0 PL=0
MOVL C01081 V=800.0 PL=0
MOVL C01082 V=800.0 PL=0
MOVL C01083 V=800.0 PL=0
MOVL C01084 V=800.0 PL=0
MOVL C01085 V=800.0 PL=0
MOVL C01086 V=800.0 PL=0
MOVL C01087 V=800.0 PL=0
MOVL C01088 V=800.0 PL=0
MOVL C01089 V=800.0 PL=0
MOVL C01090 V=800.0 PL=0
MOVL C01091 V=800.0 PL=0
MOVL C01092 V=800.0 PL=0
MOVL C01093 V=800.0 PL=0
MOVL C01094 V=800.0 PL=0
MOVL C01095 V=800.0 PL=0
MOVL C01096 V=800.0 PL=0
MOVL C01097 V=800.0 PL=0
MOVL C01098 V=800.0 PL=0
MOVL C01099 V=800.0 PL=0
MOVL C01100 V=800.0 PL=0
MOVL C01101 V=800.0 PL=0
MOVL C01102 V=800.0 PL=0
MOVL C01103 V=800.0 PL=0
MOVL C01104 V=800.0 PL=0
MOVL C01105 V=800.0 PL=0
MOVL C01106 V=800.0 PL=0
MOVL C01107 V=800.0 PL=0
MOVL C01108 V=800.0 PL=0
MOVL C01109 V=800.0 PL=0
MOVL C01110 V=800.0 PL=0
MOVL C01111 V=800.0 PL=0
MOVL C01112 V=800.0 PL=0
MOVL C01113 V=800.0 PL=0
MOVL C01114 V=800.0 PL=0
MOVL C01115 V=800.0 PL=0
MOVL C01116 V=800.0 PL=0
MOVL C01117 V=800.0 PL=0
MOVL C01118 V=800.0 PL=0
MOVL C01119 V=800.0 PL=0
MOVL C01120 V=800.0 PL=0
MOVL C01121 V=800.0 PL=0
MOVL C01122 V=800.0 PL=0
MOVL C01123 V=800.0 PL=0
MOVL C01124 V=800.0 PL=0
MOVL C01125 V=800.0 PL=0
MOVL C01126 V=800.0 PL=0
MOVL C01127 V=800.0 PL=0
MOVL C01128 V=800.0 PL=0
MOVL C01129 V=800.0 PL=0
MOVL C01130 V=800.0 PL=0
MOVL C01131 V=800.0 PL=0
MOVL C01132 V=800.0 PL=0
MOVL C01133 V=800.0 PL=0
MOVL C01134 V=800.0 PL=0
MOVL C01135 V=800.0 PL=0
MOVL C01136 V=800.0 PL=0
MOVL C01137 V=800.0 PL=0
MOVL C01138 V=800.0 PL=0
MOVL C01139 V=800.0 PL=0
MOVL C01140 V=800.0 PL=0
MOVL C01141 V=800.0 PL=0
MOVL C01142 V=800.0 PL=0
MOVL C01143 V=800.0 PL=0
MOVL C01144 V=800.0 PL=0
MOVL C01145 V=800.0 PL=0
MOVL C01146 V=800.0 PL=0
MOVL C01147 V=800.0 PL=0
MOVL C01148 V=800.0 PL=0
MOVL C01149 V=800.0 PL=0
MOVL C01150 V=800.0 PL=0
MOVL C01151 V=800.0 PL=0
MOVL C01152 V=800.0 PL=0
MOVL C01153 V=800.0 PL=0
MOVL C01154 V=800.0 PL=0
MOVL C01155 V=800.0 PL=0
MOVL C01156 V=800.0 PL=0
MOVL C01157 V=800.0 PL=0
MOVL C01158 V=800.0 PL=0
MOVL C01159 V=800.0 PL=0
MOVL C01160 V=800.0 PL=0
MOVL C01161 V=800.0 PL=0
MOVL C01162 V=800.0 PL=0
MOVL C01163 V=800.0 PL=0
MOVL C01164 V=800.0 PL=0
MOVL C01165 V=800.0 PL=0
MOVL C01166 V=800.0 PL=0
MOVL C01167 V=800.0 PL=0
MOVL C01168 V=800.0 PL=0
MOVL C01169 V=800.0 PL=0
MOVL C01170 V=800.0 PL=0
MOVL C01171 V=800.0 PL=0
MOVL C01172 V=800.0 PL=0
MOVL C01173 V=800.0 PL=0
MOVL C01174 V=800.0 PL=0
MOVL C01175 V=800.0 PL=0
MOVL C01176 V=800.0 PL=0
MOVL C01177 V=800.0 PL=0
MOVL C01178 V=800.0 PL=0
MOVL C01179 V=800.0 PL=0
MOVL C01180 V=800.0 PL=0
MOVL C01181 V=800.0 PL=0
MOVL C01182 V=800.0 PL=0
MOVL C01183 V=800.0 PL=0
MOVL C01184 V=800.0 PL=0
MOVL C01185 V=800.0 PL=0
MOVL C01186 V=800.0 PL=0
MOVL C01187 V=800.0 PL=0
MOVL C01188 V=800.0 PL=0
MOVL C01189 V=800.0 PL=0
MOVL C01190 V=800.0 PL=0
MOVL C01191 V=800.0 PL=0
MOVL C01192 V=800.0 PL=0
MOVL C01193 V=800.0 PL=0
MOVL C01194 V=800.0 PL=0
MOVL C01195 V=800.0 PL=0
MOVL C01196 V=800.0 PL=0
MOVL C01197 V=800.0 PL=0
MOVL C01198 V=800.0 PL=0
MOVL C01199 V=800.0 PL=0
MOVL C01200 V=800.0 PL=0
MOVL C01201 V=800.0 PL=0
MOVL C01202 V=800.0 PL=0
MOVL C01203 V=800.0 PL=0
MOVL C01204 V=800.0 PL=0
MOVL C01205 V=800.0 PL=0
MOVL C01206 V=800.0 PL=0
MOVL C01207 V=800.0 PL=0
MOVL C01208 V=800.0 PL=0
MOVL C01209 V=800.0 PL=0
MOVL C01210 V=800.0 PL=0
MOVL C01211 V=800.0 PL=0
MOVL C01212 V=800.0 PL=0
MOVL C01213 V=800.0 PL=0
MOVL C01214 V=800.0 PL=0
MOVL C01215 V=800.0 PL=0
MOVL C01216 V=800.0 PL=0
MOVL C01217 V=800.0 PL=0
MOVL C01218 V=800.0 PL=0
MOVL C01219 V=800.0 PL=0
MOVL C01220 V=800.0 PL=0
MOVL C01221 V=800.0 PL=0
MOVL C01222 V=800.0 PL=0
MOVL C01223 V=800.0 PL=0
MOVL C01224 V=800.0 PL=0
MOVL C01225 V=800.0 PL=0
MOVL C01226 V=800.0 PL=0
MOVL C01227 V=800.0 PL=0
MOVL C01228 V=800.0 PL=0
MOVL C01229 V=800.0 PL=0
MOVL C01230 V=800.0 PL=0
MOVL C01231 V=800.0 PL=0
MOVL C01232 V=800.0 PL=0
MOVL C01233 V=800.0 PL=0
MOVL C01234 V=800.0 PL=0
MOVL C01235 V=800.0 PL=0
MOVL C01236 V=800.0 PL=0
MOVL C01237 V=800.0 PL=0
MOVL C01238 V=800.0 PL=0
MOVL C01239 V=800.0 PL=0
MOVL C01240 V=800.0 PL=0
MOVL C01241 V=800.0 PL=0
MOVL C01242 V=800.0 PL=0
MOVL C01243 V=800.0 PL=0
MOVL C01244 V=800.0 PL=0
MOVL C01245 V=800.0 PL=0
MOVL C01246 V=800.0 PL=0
MOVL C01247 V=800.0 PL=0
MOVL C01248 V=800.0 PL=0
MOVL C01249 V=800.0 PL=0
MOVL C01250 V=800.0 PL=0
MOVL C01251 V=800.0 PL=0
MOVL C01252 V=800.0 PL=0
MOVL C01253 V=800.0 PL=0
MOVL C01254 V=800.0 PL=0
MOVL C01255 V=800.0 PL=0
MOVL C01256 V=800.0 PL=0
MOVL C01257 V=800.0 PL=0
MOVL C01258 V=800.0 PL=0
MOVL C01259 V=800.0 PL=0
MOVL C01260 V=800.0 PL=0
MOVL C01261 V=800.0 PL=0
MOVL C01262 V=800.0 PL=0
MOVL C01263 V=800.0 PL=0
MOVL C01264 V=800.0 PL=0
MOVL C01265 V=800.0 PL=0
MOVL C01266 V=800.0 PL=0
MOVL C01267 V=800.0 PL=0
MOVL C01268 V=800.0 PL=0
MOVL C01269 V=800.0 PL=0
MOVL C01270 V=800.0 PL=0
MOVL C01271 V=800.0 PL=0
MOVL C01272 V=800.0 PL=0
MOVL C01273 V=800.0 PL=0
MOVL C01274 V=800.0 PL=0
MOVL C01275 V=800.0 PL=0
MOVL C01276 V=800.0 PL=0
MOVL C01277 V=800.0 PL=0
MOVL C01278 V=800.0 PL=0
MOVL C01279 V=800.0 PL=0
MOVL C01280 V=800.0 PL=0
MOVL C01281 V=800.0 PL=0
MOVL C01282 V=800.0 PL=0
MOVL C01283 V=800.0 PL=0
MOVL C01284 V=800.0 PL=0
MOVL C01285 V=800.0 PL=0
MOVL C01286 V=800.0 PL=0
MOVL C01287 V=800.0 PL=0
MOVL C01288 V=800.0 PL=0
MOVL C01289 V=800.0 PL=0
MOVL C01290 V=800.0 PL=0
MOVL C01291 V=800.0 PL=0
MOVL C01292 V=800.0 PL=0
MOVL C01293 V=800.0 PL=0
MOVL C01294 V=800.0 PL=0
MOVL C01295 V=800.0 PL=0
MOVL C01296 V=800.0 PL=0
MOVL C01297 V=800.0 PL=0
MOVL C01298 V=800.0 PL=0
MOVL C01299 V=800.0 PL=0
MOVL C01300 V=800.0 PL=0
MOVL C01301 V=800.0 PL=0
MOVL C01302 V=800.0 PL=0
MOVL C01303 V=800.0 PL=0
MOVL C01304 V=800.0 PL=0
MOVL C01305 V=800.0 PL=0
MOVL C01306 V=800.0 PL=0
MOVL C01307 V=800.0 PL=0
MOVL C01308 V=800.0 PL=0
MOVL C01309 V=800.0 PL=0
MOVL C01310 V=800.0 PL=0
MOVL C01311 V=800.0 PL=0
MOVL C01312 V=800.0 PL=0
MOVL C01313 V=800.0 PL=0
MOVL C01314 V=800.0 PL=0
MOVL C01315 V=800.0 PL=0
MOVL C01316 V=800.0 PL=0
MOVL C01317 V=800.0 PL=0
MOVL C01318 V=800.0 PL=0
MOVL C01319 V=800.0 PL=0
MOVL C01320 V=800.0 PL=0
MOVL C01321 V=800.0 PL=0
MOVL C01322 V=800.0 PL=0
MOVL C01323 V=800.0 PL=0
MOVL C01324 V=800.0 PL=0
MOVL C01325 V=800.0 PL=0
MOVL C01326 V=800.0 PL=0
MOVL C01327 V=800.0 PL=0
MOVL C01328 V=800.0 PL=0
MOVL C01329 V=800.0 PL=0
MOVL C01330 V=800.0 PL=0
MOVL C01331 V=800.0 PL=0
MOVL C01332 V=800.0 PL=0
MOVL C01333 V=800.0 PL=0
MOVL C01334 V=800.0 PL=0
MOVL C01335 V=800.0 PL=0
MOVL C01336 V=800.0 PL=0
MOVL C01337 V=800.0 PL=0
MOVL C01338 V=800.0 PL=0
MOVL C01339 V=800.0 PL=0
MOVL C01340 V=800.0 PL=0
MOVL C01341 V=800.0 PL=0
MOVL C01342 V=800.0 PL=0
MOVL C01343 V=800.0 PL=0
MOVL C01344 V=800.0 PL=0
MOVL C01345 V=800.0 PL=0
MOVL C01346 V=800.0 PL=0
MOVL C01347 V=800.0 PL=0
MOVL C01348 V=800.0 PL=0
MOVL C01349 V=800.0 PL=0
MOVL C01350 V=800.0 PL=0
MOVL C01351 V=800.0 PL=0
MOVL C01352 V=800.0 PL=0
MOVL C01353 V=800.0 PL=0
MOVL C01354 V=800.0 PL=0
MOVL C01355 V=800.0 PL=0
MOVL C01356 V=800.0 PL=0
MOVL C01357 V=800.0 PL=0
MOVL C01358 V=800.0 PL=0
MOVL C01359 V=800.0 PL=0
MOVL C01360 V=800.0 PL=0
MOVL C01361 V=800.0 PL=0
MOVL C01362 V=800.0 PL=0
MOVL C01363 V=800.0 PL=0
MOVL C01364 V=800.0 PL=0
MOVL C01365 V=800.0 PL=0
MOVL C01366 V=800.0 PL=0
MOVL C01367 V=800.0 PL=0
MOVL C01368 V=800.0 PL=0
MOVL C01369 V=800.0 PL=0
MOVL C01370 V=800.0 PL=0
MOVL C01371 V=800.0 PL=0
MOVL C01372 V=800.0 PL=0
MOVL C01373 V=800.0 PL=0
MOVL C01374 V=800.0 PL=0
MOVL C01375 V=800.0 PL=0
MOVL C01376 V=800.0 PL=0
MOVL C01377 V=800.0 PL=0
MOVL C01378 V=800.0 PL=0
MOVL C01379 V=800.0 PL=0
MOVL C01380 V=800.0 PL=0
MOVL C01381 V=800.0 PL=0
MOVL C01382 V=800.0 PL=0
MOVL C01383 V=800.0 PL=0
MOVL C01384 V=800.0 PL=0
MOVL C01385 V=800.0 PL=0
MOVL C01386 V=800.0 PL=0
MOVL C01387 V=800.0 PL=0
MOVL C01388 V=800.0 PL=0
MOVL C01389 V=800.0 PL=0
MOVL C01390 V=800.0 PL=0
MOVL C01391 V=800.0 PL=0
MOVL C01392 V=800.0 PL=0
MOVL C01393 V=800.0 PL=0
MOVL C01394 V=800.0 PL=0
MOVL C01395 V=800.0 PL=0
MOVL C01396 V=800.0 PL=0
MOVL C01397 V=800.0 PL=0
MOVL C01398 V=800.0 PL=0
MOVL C01399 V=800.0 PL=0
MOVL C01400 V=800.0 PL=0
MOVL C01401 V=800.0 PL=0
MOVL C01402 V=800.0 PL=0
MOVL C01403 V=800.0 PL=0
MOVL C01404 V=800.0 PL=0
MOVL C01405 V=800.0 PL=0
MOVL C01406 V=800.0 PL=0
MOVL C01407 V=800.0 PL=0
MOVL C01408 V=800.0 PL=0
MOVL C01409 V=800.0 PL=0
MOVL C01410 V=800.0 PL=0
MOVL C01411 V=800.0 PL=0
MOVL C01412 V=800.0 PL=0
MOVL C01413 V=800.0 PL=0
MOVL C01414 V=800.0 PL=0
MOVL C01415 V=800.0 PL=0
MOVL C01416 V=800.0 PL=0
MOVL C01417 V=800.0 PL=0
MOVL C01418 V=800.0 PL=0
MOVL C01419 V=800.0 PL=0
MOVL C01420 V=800.0 PL=0
MOVL C01421 V=800.0 PL=0
MOVL C01422 V=800.0 PL=0
MOVL C01423 V=800.0 PL=0
MOVL C01424 V=800.0 PL=0
MOVL C01425 V=800.0 PL=0
MOVL C01426 V=800.0 PL=0
MOVL C01427 V=800.0 PL=0
MOVL C01428 V=800.0 PL=0
MOVL C01429 V=800.0 PL=0
MOVL C01430 V=800.0 PL=0
MOVL C01431 V=800.0 PL=0
MOVL C01432 V=800.0 PL=0
MOVL C01433 V=800.0 PL=0
MOVL C01434 V=800.0 PL=0
MOVL C01435 V=800.0 PL=0
MOVL C01436 V=800.0 PL=0
MOVL C01437 V=800.0 PL=0
MOVL C01438 V=800.0 PL=0
MOVL C01439 V=800.0 PL=0
MOVL C01440 V=800.0 PL=0
MOVL C01441 V=800.0 PL=0
MOVL C01442 V=800.0 PL=0
MOVL C01443 V=800.0 PL=0
MOVL C01444 V=800.0 PL=0
MOVL C01445 V=800.0 PL=0
MOVL C01446 V=800.0 PL=0
MOVL C01447 V=800.0 PL=0
MOVL C01448 V=800.0 PL=0
MOVL C01449 V=800.0 PL=0
MOVL C01450 V=800.0 PL=0
MOVL C01451 V=800.0 PL=0
MOVL C01452 V=800.0 PL=0
MOVL C01453 V=800.0 PL=0
MOVL C01454 V=800.0 PL=0
MOVL C01455 V=800.0 PL=0
MOVL C01456 V=800.0 PL=0
MOVL C01457 V=800.0 PL=0
MOVL C01458 V=800.0 PL=0
MOVL C01459 V=800.0 PL=0
MOVL C01460 V=800.0 PL=0
MOVL C01461 V=800.0 PL=0
MOVL C01462 V=800.0 PL=0
MOVL C01463 V=800.0 PL=0
MOVL C01464 V=800.0 PL=0
MOVL C01465 V=800.0 PL=0
MOVL C01466 V=800.0 PL=0
MOVL C01467 V=800.0 PL=0
MOVL C01468 V=800.0 PL=0
MOVL C01469 V=800.0 PL=0
MOVL C01470 V=800.0 PL=0
MOVL C01471 V=800.0 PL=0
MOVL C01472 V=800.0 PL=0
MOVL C01473 V=800.0 PL=0
MOVL C01474 V=800.0 PL=0
MOVL C01475 V=800.0 PL=0
MOVL C01476 V=800.0 PL=0
MOVL C01477 V=800.0 PL=0
MOVL C01478 V=800.0 PL=0
MOVL C01479 V=800.0 PL=0
MOVL C01480 V=800.0 PL=0
MOVL C01481 V=800.0 PL=0
MOVL C01482 V=800.0 PL=0
MOVL C01483 V=800.0 PL=0
MOVL C01484 V=800.0 PL=0
MOVL C01485 V=800.0 PL=0
MOVL C01486 V=800.0 PL=0
MOVL C01487 V=800.0 PL=0
MOVL C01488 V=800.0 PL=0
MOVL C01489 V=800.0 PL=0
MOVL C01490 V=800.0 PL=0
MOVL C01491 V=800.0 PL=0
MOVL C01492 V=800.0 PL=0
MOVL C01493 V=800.0 PL=0
MOVL C01494 V=800.0 PL=0
MOVL C01495 V=800.0 PL=0
MOVL C01496 V=800.0 PL=0
MOVL C01497 V=800.0 PL=0
MOVL C01498 V=800.0 PL=0
MOVL C01499 V=800.0 PL=0
MOVL C01500 V=800.0 PL=0
MOVL C01501 V=800.0 PL=0
MOVL C01502 V=800.0 PL=0
MOVL C01503 V=800.0 PL=0
MOVL C01504 V=800.0 PL=0
MOVL C01505 V=800.0 PL=0
MOVL C01506 V=800.0 PL=0
MOVL C01507 V=800.0 PL=0
MOVL C01508 V=800.0 PL=0
MOVL C01509 V=800.0 PL=0
MOVL C01510 V=800.0 PL=0
MOVL C01511 V=800.0 PL=0
MOVL C01512 V=800.0 PL=0
MOVL C01513 V=800.0 PL=0
MOVL C01514 V=800.0 PL=0
MOVL C01515 V=800.0 PL=0
MOVL C01516 V=800.0 PL=0
MOVL C01517 V=800.0 PL=0
MOVL C01518 V=800.0 PL=0
MOVL C01519 V=800.0 PL=0
MOVL C01520 V=800.0 PL=0
MOVL C01521 V=800.0 PL=0
MOVL C01522 V=800.0 PL=0
MOVL C01523 V=800.0 PL=0
MOVL C01524 V=800.0 PL=0
MOVL C01525 V=800.0 PL=0
MOVL C01526 V=800.0 PL=0
MOVL C01527 V=800.0 PL=0
MOVL C01528 V=800.0 PL=0
MOVL C01529 V=800.0 PL=0
MOVL C01530 V=800.0 PL=0
MOVL C01531 V=800.0 PL=0
MOVL C01532 V=800.0 PL=0
MOVL C01533 V=800.0 PL=0
MOVL C01534 V=800.0 PL=0
MOVL C01535 V=800.0 PL=0
MOVL C01536 V=800.0 PL=0
MOVL C01537 V=800.0 PL=0
MOVL C01538 V=800.0 PL=0
MOVL C01539 V=800.0 PL=0
MOVL C01540 V=800.0 PL=0
MOVL C01541 V=800.0 PL=0
MOVL C01542 V=800.0 PL=0
MOVL C01543 V=800.0 PL=0
MOVL C01544 V=800.0 PL=0
MOVL C01545 V=800.0 PL=0
MOVL C01546 V=800.0 PL=0
MOVL C01547 V=800.0 PL=0
MOVL C01548 V=800.0 PL=0
MOVL C01549 V=800.0 PL=0
MOVL C01550 V=800.0 PL=0
MOVL C01551 V=800.0 PL=0
MOVL C01552 V=800.0 PL=0
MOVL C01553 V=800.0 PL=0
MOVL C01554 V=800.0 PL=0
MOVL C01555 V=800.0 PL=0
MOVL C01556 V=800.0 PL=0
MOVL C01557 V=800.0 PL=0
MOVL C01558 V=800.0 PL=0
MOVL C01559 V=800.0 PL=0
MOVL C01560 V=800.0 PL=0
MOVL C01561 V=800.0 PL=0
MOVL C01562 V=800.0 PL=0
MOVL C01563 V=800.0 PL=0
MOVL C01564 V=800.0 PL=0
MOVL C01565 V=800.0 PL=0
MOVL C01566 V=800.0 PL=0
MOVL C01567 V=800.0 PL=0
MOVL C01568 V=800.0 PL=0
MOVL C01569 V=800.0 PL=0
MOVL C01570 V=800.0 PL=0
MOVL C01571 V=800.0 PL=0
MOVL C01572 V=800.0 PL=0
MOVL C01573 V=800.0 PL=0
MOVL C01574 V=800.0 PL=0
MOVL C01575 V=800.0 PL=0
MOVL C01576 V=800.0 PL=0
MOVL C01577 V=800.0 PL=0
MOVL C01578 V=800.0 PL=0
MOVL C01579 V=800.0 PL=0
MOVL C01580 V=800.0 PL=0
MOVL C01581 V=800.0 PL=0
MOVL C01582 V=800.0 PL=0
MOVL C01583 V=800.0 PL=0
MOVL C01584 V=800.0 PL=0
MOVL C01585 V=800.0 PL=0
MOVL C01586 V=800.0 PL=0
MOVL C01587 V=800.0 PL=0
MOVL C01588 V=800.0 PL=0
MOVL C01589 V=800.0 PL=0
MOVL C01590 V=800.0 PL=0
MOVL C01591 V=800.0 PL=0
MOVL C01592 V=800.0 PL=0
MOVL C01593 V=800.0 PL=0
MOVL C01594 V=800.0 PL=0
MOVL C01595 V=800.0 PL=0
MOVL C01596 V=800.0 PL=0
MOVL C01597 V=800.0 PL=0
MOVL C01598 V=800.0 PL=0
MOVL C01599 V=800.0 PL=0
MOVL C01600 V=800.0 PL=0
MOVL C01601 V=800.0 PL=0
MOVL C01602 V=800.0 PL=0
MOVL C01603 V=800.0 PL=0
MOVL C01604 V=800.0 PL=0
MOVL C01605 V=800.0 PL=0
MOVL C01606 V=800.0 PL=0
MOVL C01607 V=800.0 PL=0
MOVL C01608 V=800.0 PL=0
MOVL C01609 V=800.0 PL=0
MOVL C01610 V=800.0 PL=0
MOVL C01611 V=800.0 PL=0
MOVL C01612 V=800.0 PL=0
MOVL C01613 V=800.0 PL=0
MOVL C01614 V=800.0 PL=0
MOVL C01615 V=800.0 PL=0
MOVL C01616 V=800.0 PL=0
MOVL C01617 V=800.0 PL=0
MOVL C01618 V=800.0 PL=0
MOVL C01619 V=800.0 PL=0
MOVL C01620 V=800.0 PL=0
MOVL C01621 V=800.0 PL=0
MOVL C01622 V=800.0 PL=0
MOVL C01623 V=800.0 PL=0
MOVL C01624 V=800.0 PL=0
MOVL C01625 V=800.0 PL=0
MOVL C01626 V=800.0 PL=0
MOVL C01627 V=800.0 PL=0
MOVL C01628 V=800.0 PL=0
MOVL C01629 V=800.0 PL=0
MOVL C01630 V=800.0 PL=0
MOVL C01631 V=800.0 PL=0
MOVL C01632 V=800.0 PL=0
MOVL C01633 V=800.0 PL=0
MOVL C01634 V=800.0 PL=0
MOVL C01635 V=800.0 PL=0
MOVL C01636 V=800.0 PL=0
MOVL C01637 V=800.0 PL=0
MOVL C01638 V=800.0 PL=0
MOVL C01639 V=800.0 PL=0
MOVL C01640 V=800.0 PL=0
MOVL C01641 V=800.0 PL=0
MOVL C01642 V=800.0 PL=0
MOVL C01643 V=800.0 PL=0
MOVL C01644 V=800.0 PL=0
MOVL C01645 V=800.0 PL=0
MOVL C01646 V=800.0 PL=0
MOVL C01647 V=800.0 PL=0
MOVL C01648 V=800.0 PL=0
MOVL C01649 V=800.0 PL=0
MOVL C01650 V=800.0 PL=0
MOVL C01651 V=800.0 PL=0
MOVL C01652 V=800.0 PL=0
MOVL C01653 V=800.0 PL=0
MOVL C01654 V=800.0 PL=0
MOVL C01655 V=800.0 PL=0
MOVL C01656 V=800.0 PL=0
MOVL C01657 V=800.0 PL=0
MOVL C01658 V=800.0 PL=0
MOVL C01659 V=800.0 PL=0
MOVL C01660 V=800.0 PL=0
MOVL C01661 V=800.0 PL=0
MOVL C01662 V=800.0 PL=0
MOVL C01663 V=800.0 PL=0
MOVL C01664 V=800.0 PL=0
MOVL C01665 V=800.0 PL=0
MOVL C01666 V=800.0 PL=0
MOVL C01667 V=800.0 PL=0
MOVL C01668 V=800.0 PL=0
MOVL C01669 V=800.0 PL=0
MOVL C01670 V=800.0 PL=0
MOVL C01671 V=800.0 PL=0
MOVL C01672 V=800.0 PL=0
MOVL C01673 V=800.0 PL=0
MOVL C01674 V=800.0 PL=0
MOVL C01675 V=800.0 PL=0
MOVL C01676 V=800.0 PL=0
MOVL C01677 V=800.0 PL=0
MOVL C01678 V=800.0 PL=0
MOVL C01679 V=800.0 PL=0
MOVL C01680 V=800.0 PL=0
MOVL C01681 V=800.0 PL=0
MOVL C01682 V=800.0 PL=0
MOVL C01683 V=800.0 PL=0
MOVL C01684 V=800.0 PL=0
MOVL C01685 V=800.0 PL=0
MOVL C01686 V=800.0 PL=0
MOVL C01687 V=800.0 PL=0
MOVL C01688 V=800.0 PL=0
MOVL C01689 V=800.0 PL=0
MOVL C01690 V=800.0 PL=0
MOVL C01691 V=800.0 PL=0
MOVL C01692 V=800.0 PL=0
MOVL C01693 V=800.0 PL=0
MOVL C01694 V=800.0 PL=0
MOVL C01695 V=800.0 PL=0
MOVL C01696 V=800.0 PL=0
MOVL C01697 V=800.0 PL=0
MOVL C01698 V=800.0 PL=0
MOVL C01699 V=800.0 PL=0
MOVL C01700 V=800.0 PL=0
MOVL C01701 V=800.0 PL=0
MOVL C01702 V=800.0 PL=0
MOVL C01703 V=800.0 PL=0
MOVL C01704 V=800.0 PL=0
MOVL C01705 V=800.0 PL=0
MOVL C01706 V=800.0 PL=0
MOVL C01707 V=800.0 PL=0
MOVL C01708 V=800.0 PL=0
MOVL C01709 V=800.0 PL=0
MOVL C01710 V=800.0 PL=0
MOVL C01711 V=800.0 PL=0
MOVL C01712 V=800.0 PL=0
MOVL C01713 V=800.0 PL=0
MOVL C01714 V=800.0 PL=0
MOVL C01715 V=800.0 PL=0
MOVL C01716 V=800.0 PL=0
MOVL C01717 V=800.0 PL=0
MOVL C01718 V=800.0 PL=0
MOVL C01719 V=800.0 PL=0
MOVL C01720 V=800.0 PL=0
MOVL C01721 V=800.0 PL=0
MOVL C01722 V=800.0 PL=0
MOVL C01723 V=800.0 PL=0
MOVL C01724 V=800.0 PL=0
MOVL C01725 V=800.0 PL=0
MOVL C01726 V=800.0 PL=0
MOVL C01727 V=800.0 PL=0
MOVL C01728 V=800.0 PL=0
MOVL C01729 V=800.0 PL=0
MOVL C01730 V=800.0 PL=0
MOVL C01731 V=800.0 PL=0
MOVL C01732 V=800.0 PL=0
MOVL C01733 V=800.0 PL=0
MOVL C01734 V=800.0 PL=0
MOVL C01735 V=800.0 PL=0
MOVL C01736 V=800.0 PL=0
MOVL C01737 V=800.0 PL=0
MOVL C01738 V=800.0 PL=0
MOVL C01739 V=800.0 PL=0
MOVL C01740 V=800.0 PL=0
MOVL C01741 V=800.0 PL=0
MOVL C01742 V=800.0 PL=0
MOVL C01743 V=800.0 PL=0
MOVL C01744 V=800.0 PL=0
MOVL C01745 V=800.0 PL=0
MOVL C01746 V=800.0 PL=0
MOVL C01747 V=800.0 PL=0
MOVL C01748 V=800.0 PL=0
MOVL C01749 V=800.0 PL=0
MOVL C01750 V=800.0 PL=0
MOVL C01751 V=800.0 PL=0
MOVL C01752 V=800.0 PL=0
MOVL C01753 V=800.0 PL=0
MOVL C01754 V=800.0 PL=0
MOVL C01755 V=800.0 PL=0
MOVL C01756 V=800.0 PL=0
MOVL C01757 V=800.0 PL=0
MOVL C01758 V=800.0 PL=0
MOVL C01759 V=800.0 PL=0
MOVL C01760 V=800.0 PL=0
MOVL C01761 V=800.0 PL=0
MOVL C01762 V=800.0 PL=0
MOVL C01763 V=800.0 PL=0
MOVL C01764 V=800.0 PL=0
MOVL C01765 V=800.0 PL=0
MOVL C01766 V=800.0 PL=0
MOVL C01767 V=800.0 PL=0
MOVL C01768 V=800.0 PL=0
MOVL C01769 V=800.0 PL=0
MOVL C01770 V=800.0 PL=0
MOVL C01771 V=800.0 PL=0
MOVL C01772 V=800.0 PL=0
MOVL C01773 V=800.0 PL=0
MOVL C01774 V=800.0 PL=0
MOVL C01775 V=800.0 PL=0
MOVL C01776 V=800.0 PL=0
MOVL C01777 V=800.0 PL=0
MOVL C01778 V=800.0 PL=0
MOVL C01779 V=800.0 PL=0
MOVL C01780 V=800.0 PL=0
MOVL C01781 V=800.0 PL=0
MOVL C01782 V=800.0 PL=0
MOVL C01783 V=800.0 PL=0
MOVL C01784 V=800.0 PL=0
MOVL C01785 V=800.0 PL=0
MOVL C01786 V=800.0 PL=0
MOVL C01787 V=800.0 PL=0
MOVL C01788 V=800.0 PL=0
MOVL C01789 V=800.0 PL=0
MOVL C01790 V=800.0 PL=0
MOVL C01791 V=800.0 PL=0
MOVL C01792 V=800.0 PL=0
MOVL C01793 V=800.0 PL=0
MOVL C01794 V=800.0 PL=0
MOVL C01795 V=800.0 PL=0
MOVL C01796 V=800.0 PL=0
MOVL C01797 V=800.0 PL=0
MOVL C01798 V=800.0 PL=0
MOVL C01799 V=800.0 PL=0
MOVL C01800 V=800.0 PL=0
MOVL C01801 V=800.0 PL=0
MOVL C01802 V=800.0 PL=0
MOVL C01803 V=800.0 PL=0
MOVL C01804 V=800.0 PL=0
MOVL C01805 V=800.0 PL=0
MOVL C01806 V=800.0 PL=0
MOVL C01807 V=800.0 PL=0
MOVL C01808 V=800.0 PL=0
MOVL C01809 V=800.0 PL=0
MOVL C01810 V=800.0 PL=0
MOVL C01811 V=800.0 PL=0
MOVL C01812 V=800.0 PL=0
MOVL C01813 V=800.0 PL=0
MOVL C01814 V=800.0 PL=0
MOVL C01815 V=800.0 PL=0
MOVL C01816 V=800.0 PL=0
MOVL C01817 V=800.0 PL=0
MOVL C01818 V=800.0 PL=0
MOVL C01819 V=800.0 PL=0
MOVL C01820 V=800.0 PL=0
MOVL C01821 V=800.0 PL=0
MOVL C01822 V=800.0 PL=0
MOVL C01823 V=800.0 PL=0
MOVL C01824 V=800.0 PL=0
MOVL C01825 V=800.0 PL=0
MOVL C01826 V=800.0 PL=0
MOVL C01827 V=800.0 PL=0
MOVL C01828 V=800.0 PL=0
MOVL C01829 V=800.0 PL=0
MOVL C01830 V=800.0 PL=0
MOVL C01831 V=800.0 PL=0
MOVL C01832 V=800.0 PL=0
MOVL C01833 V=800.0 PL=0
MOVL C01834 V=800.0 PL=0
MOVL C01835 V=800.0 PL=0
MOVL C01836 V=800.0 PL=0
MOVL C01837 V=800.0 PL=0
MOVL C01838 V=800.0 PL=0
MOVL C01839 V=800.0 PL=0
MOVL C01840 V=800.0 PL=0
MOVL C01841 V=800.0 PL=0
MOVL C01842 V=800.0 PL=0
MOVL C01843 V=800.0 PL=0
MOVL C01844 V=800.0 PL=0
MOVL C01845 V=800.0 PL=0
MOVL C01846 V=800.0 PL=0
MOVL C01847 V=800.0 PL=0
MOVL C01848 V=800.0 PL=0
MOVL C01849 V=800.0 PL=0
MOVL C01850 V=800.0 PL=0
MOVL C01851 V=800.0 PL=0
MOVL C01852 V=800.0 PL=0
MOVL C01853 V=800.0 PL=0
MOVL C01854 V=800.0 PL=0
MOVL C01855 V=800.0 PL=0
MOVL C01856 V=800.0 PL=0
MOVL C01857 V=800.0 PL=0
MOVL C01858 V=800.0 PL=0
MOVL C01859 V=800.0 PL=0
MOVL C01860 V=800.0 PL=0
MOVL C01861 V=800.0 PL=0
MOVL C01862 V=800.0 PL=0
MOVL C01863 V=800.0 PL=0
MOVL C01864 V=800.0 PL=0
MOVL C01865 V=800.0 PL=0
MOVL C01866 V=800.0 PL=0
MOVL C01867 V=800.0 PL=0
MOVL C01868 V=800.0 PL=0
MOVL C01869 V=800.0 PL=0
MOVL C01870 V=800.0 PL=0
MOVL C01871 V=800.0 PL=0
MOVL C01872 V=800.0 PL=0
MOVL C01873 V=800.0 PL=0
MOVL C01874 V=800.0 PL=0
MOVL C01875 V=800.0 PL=0
MOVL C01876 V=800.0 PL=0
MOVL C01877 V=800.0 PL=0
MOVL C01878 V=800.0 PL=0
MOVL C01879 V=800.0 PL=0
MOVL C01880 V=800.0 PL=0
MOVL C01881 V=800.0 PL=0
MOVL C01882 V=800.0 PL=0
MOVL C01883 V=800.0 PL=0
MOVL C01884 V=800.0 PL=0
MOVL C01885 V=800.0 PL=0
MOVL C01886 V=800.0 PL=0
MOVL C01887 V=800.0 PL=0
MOVL C01888 V=800.0 PL=0
MOVL C01889 V=800.0 PL=0
MOVL C01890 V=800.0 PL=0
MOVL C01891 V=800.0 PL=0
MOVL C01892 V=800.0 PL=0
MOVL C01893 V=800.0 PL=0
MOVL C01894 V=800.0 PL=0
MOVL C01895 V=800.0 PL=0
MOVL C01896 V=800.0 PL=0
MOVL C01897 V=800.0 PL=0
MOVL C01898 V=800.0 PL=0
MOVL C01899 V=800.0 PL=0
MOVL C01900 V=800.0 PL=0
MOVL C01901 V=800.0 PL=0
MOVL C01902 V=800.0 PL=0
MOVL C01903 V=800.0 PL=0
MOVL C01904 V=800.0 PL=0
MOVL C01905 V=800.0 PL=0
MOVL C01906 V=800.0 PL=0
MOVL C01907 V=800.0 PL=0
MOVL C01908 V=800.0 PL=0
MOVL C01909 V=800.0 PL=0
MOVL C01910 V=800.0 PL=0
MOVL C01911 V=800.0 PL=0
MOVL C01912 V=800.0 PL=0
MOVL C01913 V=800.0 PL=0
MOVL C01914 V=800.0 PL=0
MOVL C01915 V=800.0 PL=0
MOVL C01916 V=800.0 PL=0
MOVL C01917 V=800.0 PL=0
MOVL C01918 V=800.0 PL=0
MOVL C01919 V=800.0 PL=0
MOVL C01920 V=800.0 PL=0
MOVL C01921 V=800.0 PL=0
MOVL C01922 V=800.0 PL=0
MOVL C01923 V=800.0 PL=0
MOVL C01924 V=800.0 PL=0
MOVL C01925 V=800.0 PL=0
MOVL C01926 V=800.0 PL=0
MOVL C01927 V=800.0 PL=0
MOVL C01928 V=800.0 PL=0
MOVL C01929 V=800.0 PL=0
MOVL C01930 V=800.0 PL=0
MOVL C01931 V=800.0 PL=0
MOVL C01932 V=800.0 PL=0
MOVL C01933 V=800.0 PL=0
MOVL C01934 V=800.0 PL=0
MOVL C01935 V=800.0 PL=0
MOVL C01936 V=800.0 PL=0
MOVL C01937 V=800.0 PL=0
MOVL C01938 V=800.0 PL=0
MOVL C01939 V=800.0 PL=0
MOVL C01940 V=800.0 PL=0
MOVL C01941 V=800.0 PL=0
MOVL C01942 V=800.0 PL=0
MOVL C01943 V=800.0 PL=0
MOVL C01944 V=800.0 PL=0
MOVL C01945 V=800.0 PL=0
MOVL C01946 V=800.0 PL=0
MOVL C01947 V=800.0 PL=0
MOVL C01948 V=800.0 PL=0
MOVL C01949 V=800.0 PL=0
MOVL C01950 V=800.0 PL=0
MOVL C01951 V=800.0 PL=0
MOVL C01952 V=800.0 PL=0
MOVL C01953 V=800.0 PL=0
MOVL C01954 V=800.0 PL=0
MOVL C01955 V=800.0 PL=0
MOVL C01956 V=800.0 PL=0
MOVL C01957 V=800.0 PL=0
MOVL C01958 V=800.0 PL=0
MOVL C01959 V=800.0 PL=0
MOVL C01960 V=800.0 PL=0
MOVL C01961 V=800.0 PL=0
MOVL C01962 V=800.0 PL=0
MOVL C01963 V=800.0 PL=0
MOVL C01964 V=800.0 PL=0
MOVL C01965 V=800.0 PL=0
MOVL C01966 V=800.0 PL=0
MOVL C01967 V=800.0 PL=0
MOVL C01968 V=800.0 PL=0
MOVL C01969 V=800.0 PL=0
MOVL C01970 V=800.0 PL=0
MOVL C01971 V=800.0 PL=0
MOVL C01972 V=800.0 PL=0
MOVL C01973 V=800.0 PL=0
MOVL C01974 V=800.0 PL=0
MOVL C01975 V=800.0 PL=0
MOVL C01976 V=800.0 PL=0
MOVL C01977 V=800.0 PL=0
MOVL C01978 V=800.0 PL=0
MOVL C01979 V=800.0 PL=0
MOVL C01980 V=800.0 PL=0
MOVL C01981 V=800.0 PL=0
MOVL C01982 V=800.0 PL=0
MOVL C01983 V=800.0 PL=0
MOVL C01984 V=800.0 PL=0
MOVL C01985 V=800.0 PL=0
MOVL C01986 V=800.0 PL=0
MOVL C01987 V=800.0 PL=0
MOVL C01988 V=800.0 PL=0
MOVL C01989 V=800.0 PL=0
MOVL C01990 V=800.0 PL=0
MOVL C01991 V=800.0 PL=0
MOVL C01992 V=800.0 PL=0
MOVL C01993 V=800.0 PL=0
MOVL C01994 V=800.0 PL=0
MOVL C01995 V=800.0 PL=0
MOVL C01996 V=800.0 PL=0
MOVL C01997 V=800.0 PL=0
MOVL C01998 V=800.0 PL=0
MOVL C01999 V=800.0 PL=0
MOVL C02000 V=800.0 PL=0
MOVL C02001 V=800.0 PL=0
MOVL C02002 V=800.0 PL=0
MOVL C02003 V=800.0 PL=0
MOVL C02004 V=800.0 PL=0
MOVL C02005 V=800.0 PL=0
MOVL C02006 V=800.0 PL=0
MOVL C02007 V=800.0 PL=0
MOVL C02008 V=800.0 PL=0
MOVL C02009 V=800.0 PL=0
MOVL C02010 V=800.0 PL=0
MOVL C02011 V=800.0 PL=0
MOVL C02012 V=800.0 PL=0
MOVL C02013 V=800.0 PL=0
MOVL C02014 V=800.0 PL=0
MOVL C02015 V=800.0 PL=0
MOVL C02016 V=800.0 PL=0
MOVL C02017 V=800.0 PL=0
MOVL C02018 V=800.0 PL=0
MOVL C02019 V=800.0 PL=0
MOVL C02020 V=800.0 PL=0
MOVL C02021 V=800.0 PL=0
MOVL C02022 V=800.0 PL=0
MOVL C02023 V=800.0 PL=0
MOVL C02024 V=800.0 PL=0
MOVL C02025 V=800.0 PL=0
MOVL C02026 V=800.0 PL=0
MOVL C02027 V=800.0 PL=0
MOVL C02028 V=800.0 PL=0
MOVL C02029 V=800.0 PL=0
MOVL C02030 V=800.0 PL=0
MOVL C02031 V=800.0 PL=0
MOVL C02032 V=800.0 PL=0
MOVL C02033 V=800.0 PL=0
MOVL C02034 V=800.0 PL=0
MOVL C02035 V=800.0 PL=0
MOVL C02036 V=800.0 PL=0
MOVL C02037 V=800.0 PL=0
MOVL C02038 V=800.0 PL=0
MOVL C02039 V=800.0 PL=0
MOVL C02040 V=800.0 PL=0
MOVL C02041 V=800.0 PL=0
MOVL C02042 V=800.0 PL=0
MOVL C02043 V=800.0 PL=0
MOVL C02044 V=800.0 PL=0
MOVL C02045 V=800.0 PL=0
MOVL C02046 V=800.0 PL=0
MOVL C02047 V=800.0 PL=0
MOVL C02048 V=800.0 PL=0
MOVL C02049 V=800.0 PL=0
MOVL C02050 V=800.0 PL=0
MOVL C02051 V=800.0 PL=0
MOVL C02052 V=800.0 PL=0
MOVL C02053 V=800.0 PL=0
MOVL C02054 V=800.0 PL=0
MOVL C02055 V=800.0 PL=0
MOVL C02056 V=800.0 PL=0
